// Mitsubishi GX Works2 project: GHEP-Q02U   PLC: Q02U

// global labels: Global1
VAR_GLOBAL
  Servo_Ready_T AT M1104 : BOOL;  (* Cam bien Servo Ready Truc Thu T (X0 16DT) *)
  Servo_Ready_X1 AT M1105 : BOOL;  (* Cam bien Servo Ready Truc Xa X1 (X1 16DT) *)
  Servo_Ready_X2 AT M1106 : BOOL;  (* Cam bien Servo Ready Truc Master X2 (X2 16DT) *)
  Servo_Ready_Ms AT M1107 : BOOL;  (* Cam bien Servo Ready Truc Ghep Ms (X3 16DT) *)
  Servo_Ready_S AT M1108 : BOOL;  (* Cam bien Servo Ready Truc Trang Dau S (X4 16DT) *)
  Pen1_Input_16DT AT M1109 : BOOL;  (* Tin hieu Pen 1 (X5 16DT) *)
  Pen2_Input_16DT AT M1110 : BOOL;  (* Tin hieu Pen 2 (X6 16DT) *)
  Jog_Input_16DT AT M1111 : BOOL;  (* Tin hieu Bo Cham 16DT (X7 16DT) *)
  Sensor_Rev_M AT X50 : BOOL;  (* Cam bien tiem can dem 1 vong cuon M (X50) *)
  Sensor_Rev_U AT X51 : BOOL;  (* Cam bien tiem can dem 1 vong cuon U (X51) *)
  Physical_Start_PB AT X52 : BOOL;  (* Nut nhan vat ly START QX40 (X52) *)
  Physical_Stop_PB AT X53 : BOOL;  (* Nut nhan vat ly STOP QX40 (X53) *)
  Physical_Inc_PB AT X54 : BOOL;  (* Nut nhan vat ly TANG TOC INC QX40 (X54) *)
  Physical_Dec_PB AT X55 : BOOL;  (* Nut nhan vat ly GIAM TOC DEC QX40 (X55) *)
  Pen1_Toggle_PB AT X56 : BOOL;  (* Nut nhan Toggle Pen 1 QX40 (X56) *)
  Pen2_Toggle_PB AT X57 : BOOL;  (* Nut nhan Toggle Pen 2 QX40 (X57) *)
  Switch_Hold_M AT X58 : BOOL;  (* Cong tac giu Torque Thang M khi dung (X58) *)
  Switch_Hold_U AT X59 : BOOL;  (* Cong tac giu Torque Xa U khi dung (X59) *)
  Switch_Wash_Ms AT X5A : BOOL;  (* Cong tac quay rua may bo cham Ms khi dung (X5A) *)
  Switch_Wash_S AT X5B : BOOL;  (* Cong tac quay rua may bo cham S khi dung (X5B) *)
  Physical_Jog_PB AT X5C : BOOL;  (* Nut nhan co ben ngoai BO CHAM NOI MANG QX40 (X5C) *)
  Servo_ON_T AT M1304 : BOOL;  (* Ngo ra Servo ON Truc Thu T (Y8 16DT) *)
  Servo_ON_X1 AT M1305 : BOOL;  (* Ngo ra Servo ON Truc Xa X1 (Y9 16DT) *)
  Servo_ON_X2 AT M1306 : BOOL;  (* Ngo ra Servo ON Truc Master X2 (YA 16DT) *)
  Servo_ON_Ms AT M1307 : BOOL;  (* Ngo ra Servo ON Truc Ghep Ms (YB 16DT) *)
  Servo_ON_S AT M1308 : BOOL;  (* Ngo ra Servo ON Truc Trang Dau S (YC 16DT) *)
  Pen1_Output AT M1309 : BOOL;  (* Ngo ra Ben Ep Pen 1 (YD 16DT) *)
  Pen2_Output AT M1310 : BOOL;  (* Ngo ra Ben Ep Pen 2 (YE 16DT) *)
  HMI_Auto_Mode AT M100 : BOOL;  (* Che do Auto / Manual *)
  HMI_Reset_Error AT M101 : BOOL;  (* Reset loi he thong *)
  HMI_Start AT M102 : BOOL;  (* Nut Start khoi dong HMI *)
  HMI_Stop AT M103 : BOOL;  (* Nut Stop dung may HMI *)
  HMI_Reset_Length AT M104 : BOOL;  (* Reset tong chieu dai met hang *)
  HMI_Reset_Roll_T AT M105 : BOOL;  (* Nap lai duong kinh cuon moi T *)
  HMI_Reset_Roll_M AT M106 : BOOL;  (* Nap lai duong kinh cuon moi M *)
  HMI_Reset_Roll_U AT M107 : BOOL;  (* Nap lai duong kinh cuon moi U *)
  HMI_PID_Enable AT M108 : BOOL;  (* Bat tat che do PID *)
  HMI_Inc_Hold AT M109 : BOOL;  (* Phim INC tang toc HMI *)
  HMI_Dec_Hold AT M114 : BOOL;  (* Phim DEC giam toc HMI *)
  HMI_Pen1_Cmd AT M115 : BOOL;  (* Lenh ON/OFF Pen 1 tu HMI *)
  HMI_Pen2_Cmd AT M116 : BOOL;  (* Lenh ON/OFF Pen 2 tu HMI *)
  Zero_Set_T AT M110 : BOOL;  (* Nut Set Zero Loadcell T *)
  Zero_Set_X1 AT M111 : BOOL;  (* Nut Set Zero Loadcell X1 *)
  Zero_Set_M AT M112 : BOOL;  (* Nut Set Zero Loadcell M *)
  Zero_Set_U AT M113 : BOOL;  (* Nut Set Zero Loadcell U *)
  HMI_Test_T AT M170 : BOOL;  (* Co Test chay thu rieng Truc Thu T *)
  HMI_Test_X1 AT M171 : BOOL;  (* Co Test chay thu rieng Truc Xa X1 *)
  HMI_Test_X2 AT M172 : BOOL;  (* Co Test chay thu rieng Truc Master X2 *)
  HMI_Test_Ms AT M173 : BOOL;  (* Co Test chay thu rieng Truc Ghep Ms *)
  HMI_Test_S AT M174 : BOOL;  (* Co Test chay thu rieng Truc Trang Dau S *)
  HMI_Test_M AT M175 : BOOL;  (* Co Test thu Luc Thang Tu M *)
  HMI_Test_U AT M176 : BOOL;  (* Co Test chay thu rieng Truc Xa Metalize U *)
  Calib_Set_T AT M120 : BOOL;  (* Nut Calib Span Loadcell T *)
  Calib_Set_X1 AT M121 : BOOL;  (* Nut Calib Span Loadcell X1 *)
  Calib_Set_M AT M122 : BOOL;  (* Nut Calib Span Loadcell M *)
  Calib_Set_U AT M123 : BOOL;  (* Nut Calib Span Loadcell U *)
  Servo_Not_Ready_Fault AT M134 : BOOL;  (* Co bao loi Servo Not Ready *)
  Hold_Torque_Stop_M AT M130 : BOOL;  (* Giu Torque M khi dung may *)
  Hold_Torque_Stop_U AT M131 : BOOL;  (* Giu Torque U khi dung may *)
  Anti_Dry_Rotate_S AT M132 : BOOL;  (* Bo cham S khi dung may *)
  Anti_Dry_Rotate_Ms AT M133 : BOOL;  (* Bo cham Ms khi dung may *)
  HMI_Reset_All_Rolls AT M135 : BOOL;  (* Nut thay cuon moi toan bo (Reset ca 3 cuon va xoa met) *)
  HMI_Jog_Crawl_Cmd AT M136 : BOOL;  (* Nut bo cham noi mang 2 m/p giu de chay tha de dung *)
  HMI_Cmd_Apply_Recipe AT M137 : BOOL;  (* Nut ap dung cong thuc don hang da chon *)
  HMI_Cmd_Save_Recipe AT M138 : BOOL;  (* Nut luu thong so hien tai vao cong thuc *)
  Weight_Net_T AT D510 : REAL;  (* Trong luong Luc cang thuc te T (kg/N) *)
  Weight_Net_X1 AT D512 : REAL;  (* Trong luong Luc cang thuc te X1 (kg/N) *)
  Weight_Net_M AT D514 : REAL;  (* Trong luong Luc cang thuc te M (kg/N) *)
  Weight_Net_U AT D516 : REAL;  (* Trong luong Luc cang thuc te U (kg/N) *)
  HMI_Cmd_Zero_Set AT M118 : BOOL;  (* Nut bam Set Zero chung cho truc dang chon tren HMI *)
  HMI_Cmd_Calib_Set AT M119 : BOOL;  (* Nut bam Calib Span chung cho truc dang chon tren HMI *)
  HMI_Cmd_Save_PID AT M125 : BOOL;  (* Nut bam Luu cai dat PID / Calib tren HMI *)
  HMI_Cmd_AutoTune AT M126 : BOOL;  (* Nut bam Kich hoat Auto-Tuning PID cho truc dang chon *)
  HMI_Status_AT_Busy AT M127 : BOOL;  (* Den bao dang chay Auto-Tuning *)
  HMI_Status_AT_Done AT M128 : BOOL;  (* Den bao da Auto-Tuning xong va da tu cap nhat Kp Ki Kd *)
  HMI_Status_Text_Code AT D602 : INT;  (* Ma trang thai van hanh hien thi tieng Viet tren HMI *)
  HMI_Recipe_Select AT D604 : INT;  (* Chon cong thuc don hang Recipe (1..5) *)
  HMI_Disp_Zero_Offset AT D608 : REAL;  (* O nhap Zero Offset duy nhat tren HMI *)
  HMI_Axis_Select AT D610 : INT;  (* Chon truc tren HMI (1=Thu T, 2=Xa X1, 3=Master X2, 4=Ghep Ms, 5=Dau S, 6=Thang M, 7=Xa U) *)
  HMI_Disp_Kp AT D612 : REAL;  (* O nhap Kp duy nhat tren HMI *)
  HMI_Disp_Ki AT D614 : REAL;  (* O nhap Ki duy nhat tren HMI *)
  HMI_Disp_Kd AT D616 : REAL;  (* O nhap Kd duy nhat tren HMI *)
  HMI_Disp_Calib_Gain AT D618 : REAL;  (* O nhap Calib Gain duy nhat tren HMI *)
  Gear_Ratio_T AT D620 : REAL;  (* Ty so truyen Hop so Thu T (vi du 10.1) *)
  Gear_Ratio_X1 AT D622 : REAL;  (* Ty so truyen Hop so Xa X1 (vi du 8.0) *)
  Gear_Ratio_X2 AT D624 : REAL;  (* Ty so truyen Hop so Master X2 (vi du 8.0) *)
  Gear_Ratio_Ms AT D626 : REAL;  (* Ty so truyen Hop so Ghep Ms (vi du 10.0) *)
  Gear_Ratio_S AT D628 : REAL;  (* Ty so truyen Hop so Trang Dau S (vi du 10.0) *)
  Gear_Ratio_U AT D630 : REAL;  (* Ty so truyen Hop so Xa U (vi du 1.0) *)
  Dia_X1_Roller_mm AT D638 : REAL;  (* Duong kinh lo Keo X1 (mm, vi du 300.5) *)
  Dia_Ms_Roller_mm AT D640 : REAL;  (* Duong kinh lo ghep Ms (mm, vi du 200.0) *)
  Dia_X2_Roller_mm AT D642 : REAL;  (* Duong kinh lo Master X2 (mm, vi du 300.5) *)
  Dia_S_Roller_mm AT D648 : REAL;  (* Duong kinh lo Dau S (mm, vi du 100.0) *)
  SP_Tension_T AT D660 : REAL;  (* Luc cang SP Truc T (kg) *)
  SP_Tension_X1 AT D662 : REAL;  (* Luc cang SP Truc X1 (kg) *)
  SP_Tension_M AT D664 : REAL;  (* Luc cang SP Truc M (kg) *)
  Taper_Percent_T AT D666 : REAL;  (* Ty le Con giam luc cang cuon thu T (%) *)
  SP_Tension_U AT D668 : REAL;  (* Luc cang SP Truc U (kg) *)
  Kp_T AT D670 : REAL;  (* He so Kp PID Truc T *)
  Ki_T AT D672 : REAL;  (* He so Ki PID Truc T *)
  Kd_T AT D674 : REAL;  (* He so Kd PID Truc T *)
  Kp_X1 AT D676 : REAL;  (* He so Kp PID Truc X1 *)
  Ki_X1 AT D678 : REAL;  (* He so Ki PID Truc X1 *)
  Kd_X1 AT D680 : REAL;  (* He so Kd PID Truc X1 *)
  Kp_X2 AT D682 : REAL;  (* He so Kp PID Toc do Master X2 *)
  Ki_X2 AT D684 : REAL;  (* He so Ki PID Toc do Master X2 *)
  Kd_X2 AT D686 : REAL;  (* He so Kd PID Toc do Master X2 *)
  Kp_Ms AT D688 : REAL;  (* He so Kp PID Toc do Ghep Ms *)
  Ki_Ms AT D689 : REAL;  (* He so Ki PID Toc do Ghep Ms *)
  Kd_Ms AT D692 : REAL;  (* He so Kd PID Toc do Ghep Ms *)
  Kp_S AT D694 : REAL;  (* He so Kp PID Toc do Truc S *)
  Ki_S AT D696 : REAL;  (* He so Ki PID Toc do Truc S *)
  Kd_S AT D698 : REAL;  (* He so Kd PID Toc do Truc S *)
  Set_Target_Length AT D700 : REAL;  (* Chieu dai met hang cai dat tu dung (m) *)
  Decel_Distance_Meters AT D702 : REAL;  (* Khoang cach bao giam toc truoc khi dung (m) *)
  Ramp_Accel_Rate AT D704 : REAL;  (* Thanh ghi gia toc ACC (m/p/s) *)
  Ramp_Decel_Rate AT D706 : REAL;  (* Thanh ghi giam toc DEC (m/p/s) *)
  Total_Length_Meters AT D708 : REAL;  (* Tong so met hang da ghep (m) *)
  Release_Pen_Speed_MPM AT D710 : REAL;  (* Toc do nhan bi 2 Pen ep mang (m/p) *)
  Real_Dia_U_mm AT D720 : REAL;  (* Duong kinh thuc cuon U (mm) *)
  Real_Dia_M_mm AT D722 : REAL;  (* Duong kinh thuc cuon M (mm) *)
  Real_Dia_T_mm AT D724 : REAL;  (* Duong kinh thuc cuon T (mm) *)
  Current_Line_MPM AT D730 : REAL;  (* Toc do hien tai (m/p) *)
  Target_Line_MPM AT D732 : REAL;  (* Toc do muc tieu (m/p) *)
  Max_Speed_MPM AT D734 : REAL;  (* Toc do Max (100.0 m/p) *)
  Min_Speed_MPM AT D736 : REAL;  (* Toc do Min (2.0 m/p) *)
  Anti_Dry_Crawl_Speed AT D738 : REAL;  (* Toc do bo cham rua may (1.0 m/p) *)
  Core_Dia_T_mm AT D740 : REAL;  (* Duong kinh loi cuon T (mm) *)
  Core_Dia_M_mm AT D742 : REAL;  (* Duong kinh loi cuon M (mm) *)
  Core_Dia_U_mm AT D744 : REAL;  (* Duong kinh loi cuon U (mm) *)
  Max_Dia_T_mm AT D750 : REAL;  (* Duong kinh Max cuon T (mm) *)
  Max_Dia_M_mm AT D752 : REAL;  (* Duong kinh Max cuon M (mm) *)
  Max_Dia_U_mm AT D754 : REAL;  (* Duong kinh Max cuon U (mm) *)
  Speed_Ratio_T AT D756 : REAL;  (* Ty le toc do Truc T giu Torque (vi du 1.05) *)
  Speed_Ratio_X1 AT D758 : REAL;  (* Ty le toc do Truc Xa X1 (vi du 1.00) *)
  Speed_Offset_X1 AT D760 : REAL;  (* Bu toc do Truc Xa X1 *)
  Speed_Ratio_Ms AT D762 : REAL;  (* Ty le dong bo toc do Truc Ms (vi du 1.00) *)
  Speed_Offset_Ms AT D764 : REAL;  (* Bu toc do Truc Ghep Ms *)
  Speed_Ratio_S AT D766 : REAL;  (* Ty le toc do Truc S (vi du 1.00) *)
  Speed_Offset_S AT D768 : REAL;  (* Bu toc do Truc Trang Dau S *)
  Min_Torque_M AT D770 : REAL;  (* Torque Min Thang M (%) *)
  Max_Torque_M AT D772 : REAL;  (* Torque Max Thang M (%) *)
  Init_Holding_Torque_M AT D774 : REAL;  (* Torque ban dau Thang M (%) *)
  Init_Holding_Torque_U AT D776 : REAL;  (* Torque ban dau giu cuon U (%) *)
  Min_Torque_U AT D778 : REAL;  (* Torque Min Xa U (%) *)
  Max_Torque_U AT D780 : REAL;  (* Torque Max Xa U (%) *)
  SP_Speed_S AT D782 : REAL;  (* Toc do Setpoint Truc S *)
  Feedback_Speed_S AT D784 : REAL;  (* Toc do Feedback Truc S *)
  Feedback_Speed_X2 AT D786 : REAL;  (* Toc do Feedback Master X2 *)
  Feedback_Speed_Ms AT D788 : REAL;  (* Toc do Feedback Ghep Ms *)
  Test_Speed_T AT D800 : REAL;  (* Toc do cai dat Test Truc T (0..16000) *)
  Test_Torque_T AT D802 : REAL;  (* Torque cai dat Test Truc T (0..16000) *)
  Test_Speed_X1 AT D804 : REAL;  (* Toc do cai dat Test Truc X1 (0..16000) *)
  Test_Speed_X2 AT D806 : REAL;  (* Toc do cai dat Test Truc X2 (0..16000) *)
  Test_Speed_Ms AT D808 : REAL;  (* Toc do cai dat Test Truc Ms (0..16000) *)
  Test_Speed_S AT D810 : REAL;  (* Toc do cai dat Test Truc S (0..16000) *)
  Test_Torque_M AT D812 : REAL;  (* Torque cai dat Test Thang M (0..16000) *)
  Test_Speed_U AT D814 : REAL;  (* Toc do cai dat Test Truc U (0..16000) *)
  Max_RPM_X2 AT D820 : REAL;  (* Toc do Max RPM Master X2 (1000.0) *)
  Max_RPM_X1 AT D822 : REAL;  (* Toc do Max RPM Xa X1 (1000.0) *)
  Max_RPM_Ms AT D824 : REAL;  (* Toc do Max RPM Ghep Ms (3000.0) *)
  Max_RPM_S AT D826 : REAL;  (* Toc do Max RPM Trang Dau S (3000.0) *)
  Max_RPM_T AT D828 : REAL;  (* Toc do Max RPM Thu T (1500.0) *)
  Calib_Gain_T AT D830 : REAL;  (* He so Calib Gain Loadcell T *)
  Calib_Gain_X1 AT D832 : REAL;  (* He so Calib Gain Loadcell X1 *)
  Calib_Gain_M AT D834 : REAL;  (* He so Calib Gain Loadcell M *)
  Calib_Gain_U AT D836 : REAL;  (* He so Calib Gain Loadcell U *)
  Kp_M AT D840 : REAL;  (* He so Kp PID Truc M *)
  Ki_M AT D842 : REAL;  (* He so Ki PID Truc M *)
  Kd_M AT D844 : REAL;  (* He so Kd PID Truc M *)
  Kp_U AT D846 : REAL;  (* He so Kp PID Truc U *)
  Ki_U AT D848 : REAL;  (* He so Ki PID Truc U *)
  Kd_U AT D850 : REAL;  (* He so Kd PID Truc U *)
  Zero_Offset_T AT D852 : REAL;  (* Diem 0 Zero Offset Loadcell Thu T *)
  Zero_Offset_X1 AT D854 : REAL;  (* Diem 0 Zero Offset Loadcell Xa X1 *)
  Zero_Offset_M AT D856 : REAL;  (* Diem 0 Zero Offset Thang Tu Metalize M *)
  Zero_Offset_U AT D858 : REAL;  (* Diem 0 Zero Offset Cuon Xa Sau Cung U *)
  CCLink_AD_Avg_Mode AT D860 : WORD;  (* Che do lay trung binh BFM 0 64AD (H3333=Moving Avg) *)
  CCLink_AD_Avg_CH1 AT D861 : INT;  (* So mau trung binh CH1 BFM 1 (Loadcell Thu T) *)
  CCLink_AD_Avg_CH2 AT D862 : INT;  (* So mau trung binh CH2 BFM 2 (Loadcell Xa X1) *)
  CCLink_AD_Avg_CH3 AT D863 : INT;  (* So mau trung binh CH3 BFM 3 (Loadcell Thang M) *)
  CCLink_AD_Avg_CH4 AT D864 : INT;  (* So mau trung binh CH4 BFM 4 (Loadcell Xa U) *)
  CCLink_AD_Conv_En AT D865 : INT;  (* Cho phep chuyen doi AD 4 kenh BFM 10 (0=Enable) *)
END_VAR

// task Task_01 (event TRUE, interval 0, priority 31): POU_01
// task POU_INIT (event TRUE, interval 0, priority 31): POU_INIT

PROGRAM POU_01
VAR
  pid_T : FB_TENSION_PID;  (* Instance PID Luc cang Thu T *)
  pid_X1 : FB_TENSION_PID;  (* Instance PID Luc cang Xa X1 *)
  pid_M : FB_TENSION_PID;  (* Instance PID Thang Tu M *)
  pid_U : FB_TENSION_PID;  (* Instance PID Luc cang Xa U *)
  pid_X2 : FB_TENSION_PID;  (* Instance PID Toc do Master X2 *)
  pid_Ms : FB_TENSION_PID;  (* Instance PID Toc do Ghep Ms *)
  pid_S : FB_TENSION_PID;  (* Instance PID Toc do Trang Dau S *)
  fbCCLink : FFB_CCLINK_CONTROL;  (* Instance Control CC-Link Master *)
  Base_Speed_X2 : REAL;  (* Toc do nen Master X2 *)
  SP_Speed_X2 : REAL;  (* Toc do Setpoint Master X2 *)
  SP_Speed_X1 : REAL;  (* Toc do Setpoint Xa X1 *)
  SP_Speed_Ms : REAL;  (* Toc do Setpoint Ghep Ms *)
  SP_Speed_T : REAL;  (* Toc do Setpoint Thu T *)
  Calc_Speed_X2 : REAL;  (* Toc do tinh toan Master X2 *)
  Calc_Speed_T : REAL;  (* Toc do tinh toan Thu T *)
  Calc_Torque_T : REAL;  (* Torque tinh toan Thu T *)
  Calc_Speed_X1 : REAL;  (* Toc do tinh toan Xa X1 *)
  Calc_Speed_Ms : REAL;  (* Toc do tinh toan Ghep Ms *)
  Calc_Speed_S : REAL;  (* Toc do tinh toan Trang Dau S *)
  Calc_Speed_U : REAL;  (* Toc do tinh toan Xa U *)
  Calc_Torque_M : REAL;  (* Torque tinh toan Thang M *)
  Base_Torque_M : REAL;  (* Torque nen co ban Thang M *)
  State_Machine : DINT;  (* Trang thai van hanh State Machine *)
  ADC_CH1_Val : WORD;  (* Bien tam doc ADC CH1 *)
  ADC_CH2_Val : WORD;  (* Bien tam doc ADC CH2 *)
  ADC_CH3_Val : WORD;  (* Bien tam doc ADC CH3 *)
  ADC_CH4_Val : WORD;  (* Bien tam doc ADC CH4 *)
  Effective_SP_T : REAL;  (* Luc cang SP cuon T sau khi tinh Con luc Taper *)
  Auto_Decel_Flag : BOOL;  (* Co tu dong giam toc khi sap dat tong chieu dai *)
  ADC_Filter_T : REAL;  (* Bo loc nhieu trung binh dong Loadcell T *)
  ADC_Filter_X1 : REAL;  (* Bo loc nhieu trung binh dong Loadcell X1 *)
  ADC_Filter_M : REAL;  (* Bo loc nhieu trung binh dong Loadcell M *)
  ADC_Filter_U : REAL;  (* Bo loc nhieu trung binh dong Loadcell U *)
  Cmd_Start : BOOL;  (* Lenh Tong Start (HMI + Nut vat ly X52) *)
  Cmd_Stop : BOOL;  (* Lenh Tong Stop (HMI + Nut vat ly X53) *)
  Cmd_Inc : BOOL;  (* Lenh Tong INC Tang toc (HMI + Nut vat ly X54) *)
  Cmd_Dec : BOOL;  (* Lenh Tong DEC Giam toc (HMI + Nut vat ly X55) *)
  Cmd_Jog_Crawl : BOOL;  (* Lenh Tong Bo cham noi mang 2 m/p (HMI + Nut co X5C) *)
  Inc_Hold_Timer : DINT;  (* Timer bam giu phim Tang toc INC *)
  Dec_Hold_Timer : DINT;  (* Timer bam giu phim Giam toc DEC *)
  Curr_Pulse_T : DINT;  (* Xung Encoder Thu T *)
  Last_Pulse_T : DINT;  (* Xung Encoder Thu T vong truoc *)
  Curr_Pulse_X2 : DINT;  (* Xung Encoder Master X2 *)
  Last_Pulse_X2_T : DINT;  (* Xung Master X2 khi Thu T quay 1 vong *)
  Last_Pulse_X2_M : DINT;  (* Xung Master X2 khi Cuon M quay 1 vong *)
  Last_Pulse_X2_U : DINT;  (* Xung Master X2 khi Cuon U quay 1 vong *)
  Last_Pulse_X2_Len : DINT;  (* Xung Master X2 vong truoc de do met *)
  Delta_Pulse_X2 : DINT;  (* So xung Master X2 tang them moi chu ky *)
  Delta_Length_mm : REAL;  (* So mm mang tang them moi chu ky *)
  Accum_Length_mm : REAL;  (* Tich luy mm mang de doi ra met *)
  Trig_X50 : BOOL;  (* Xung phat hien cam bien X50 cuon M *)
  Trig_X51 : BOOL;  (* Xung phat hien cam bien X51 cuon U *)
  Prev_X50 : BOOL;  (* Trang thai X50 vong scan truoc *)
  Prev_X51 : BOOL;  (* Trang thai X51 vong scan truoc *)
  Raw_Dia_T_mm : REAL;  (* Duong kinh tho tinh duoc cuon T *)
  Raw_Dia_M_mm : REAL;  (* Duong kinh tho tinh duoc cuon M *)
  Raw_Dia_U_mm : REAL;  (* Duong kinh tho tinh duoc cuon U *)
  Rev_Count_T : DINT;  (* So vong quay cuon T *)
  Rev_Count_M : DINT;  (* So vong quay cuon M *)
  Rev_Count_U : DINT;  (* So vong quay cuon U *)
  Dynamic_Accel_Step : REAL;  (* Buoc gia toc dong tang giam luy tien *)
  Trig_Pen1 : BOOL;  (* Xung nhan phim Toggle Pen 1 X56 *)
  Trig_Pen2 : BOOL;  (* Xung nhan phim Toggle Pen 2 X57 *)
  Prev_Pen1_PB : BOOL;  (* Trang thai X56 vong scan truoc *)
  Prev_Pen2_PB : BOOL;  (* Trang thai X57 vong scan truoc *)
  Prev_Pen1_16DT : BOOL;  (* Trang thai Pen 1 tren 16DT vong truoc *)
  Prev_Pen2_16DT : BOOL;  (* Trang thai Pen 2 tren 16DT vong truoc *)
  Pen1_State : BOOL;  (* Trang thai ON/OFF hien tai Pen 1 *)
  Pen2_State : BOOL;  (* Trang thai ON/OFF hien tai Pen 2 *)
  PID_Out_T : REAL;  (* Output PID sau khi lay tu pid_T *)
  PID_Out_X1 : REAL;  (* Output PID sau khi lay tu pid_X1 *)
  PID_Out_M : REAL;  (* Output PID sau khi lay tu pid_M *)
  PID_Out_U : REAL;  (* Output PID sau khi lay tu pid_U *)
  PID_Out_X2 : REAL;  (* Output PID Toc do X2 *)
  PID_Out_Ms : REAL;  (* Output PID Toc do Ms *)
  PID_Out_S : REAL;  (* Output PID Toc do S *)
  Trig_PID_10ms : BOOL;  (* Xung kich hoat PID moi 10ms (SM409) *)
  Prev_SM409 : BOOL;  (* Trang thai SM409 vong scan truoc *)
  Pen_Auto_Engaged : BOOL;  (* Co tu dong kep 2 Pen khi toc do vuot 5 m/p *)
  Prev_Recipe_Select : INT;  (* Luu gia tri Recipe da chon vong scan truoc *)
END_VAR
(* ============================================================================ *)
(* MÃ NGUỒN POU_01: HỆ THỐNG MÁY GHÉP MÀNG METALIZE TỰ ĐỘNG - MITSUBISHI Q02U  *)
(* ĐỒNG BỘ VẬN TỐC DÀI THEO TRỤC CHÍNH X2 + SPEED_RATIO CHO TỪNG TRỤC           *)
(* TOÀN BỘ TÍNH TOÁN DÙNG CHUẨN SỐ THỰC FLOAT / REAL (FLOAT [Single Precision]) *)
(* ============================================================================ *)

(* 1. BẢO VỆ 5 TRỤC SERVO READY TRÊN MODULE 16DT (X0..X4 = M1136..M1140 - TRẠM 5) *)
Servo_Not_Ready_Fault := NOT(Servo_Ready_T) OR NOT(Servo_Ready_X1) OR NOT(Servo_Ready_X2) OR NOT(Servo_Ready_Ms) OR NOT(Servo_Ready_S);

IF Servo_Not_Ready_Fault AND State_Machine = 1 THEN
    State_Machine := 0; (* Dừng khẩn cấp nếu đang chạy tự động *)
END_IF;

(* 2. ĐIỀU KHIỂN CÔNG TẮC GIỮ TORQUE & BÒ CHẬM RỬA MÁY TRÊN QX40 (X58..X5B) *)
Hold_Torque_Stop_M := Switch_Hold_M;   (* X58 *)
Hold_Torque_Stop_U := Switch_Hold_U;   (* X59 *)
Anti_Dry_Rotate_Ms := Switch_Wash_Ms;  (* X5A *)
Anti_Dry_Rotate_S  := Switch_Wash_S;   (* X5B *)

(* 2.1 QUẢN LÝ CÔNG THỨC ĐƠN HÀNG (RECIPE MANAGEMENT CHO CÔNG NHÂN) *)
(* 1: Màng Mỏng 12~15mic | 2: Màng Tiêu Chuẩn 18~20mic | 3: Giấy Dày Duplex 250~350g | 4: Màng Nhôm Foil | 5: Tùy Chỉnh *)
IF HMI_Recipe_Select <= 0 OR HMI_Recipe_Select > 5 THEN
    HMI_Recipe_Select := 2; (* Mặc định chọn Recipe 2: Hàng Tiêu Chuẩn *)
END_IF;

(* TỰ ĐỘNG NẠP THÔNG SỐ KHI CÔNG NHÂN CHỌN LOẠI HÀNG HOẶC NHẤN ÁP DỤNG *)
IF (HMI_Recipe_Select <> Prev_Recipe_Select) OR HMI_Cmd_Apply_Recipe THEN
    CASE HMI_Recipe_Select OF
        1: (* 1. HÀNG MÀNG MỎNG (BOPP 12~15 mic - Bao bì bánh kẹo) *)
            Target_Line_MPM  := 45.0;  (* Tốc độ chuẩn 45 m/p *)
            SP_Tension_T     := 12.0;  (* Lực căng Thu T: 12 kg *)
            SP_Tension_X1    := 10.0;  (* Lực căng Kéo X1: 10 kg *)
            SP_Tension_M     := 4.0;   (* Lực căng Thắng Metalize M: 4 kg *)
            SP_Tension_U     := 8.0;   (* Lực căng Xả U: 8 kg *)
            Taper_Percent_T  := 15.0;  (* Giảm côn lực 15% *)
            Ramp_Accel_Rate  := 0.05;  (* Gia tốc êm ái *)
            Ramp_Decel_Rate  := 0.08;

        2: (* 2. HÀNG TIÊU CHUẨN (BOPP 18~20 mic + Giấy 100~150g - Hộp thông dụng) *)
            Target_Line_MPM  := 60.0;  (* Tốc độ chuẩn 60 m/p *)
            SP_Tension_T     := 16.0;  (* Lực căng Thu T: 16 kg *)
            SP_Tension_X1    := 14.0;  (* Lực căng Kéo X1: 14 kg *)
            SP_Tension_M     := 6.0;   (* Lực căng Thắng Metalize M: 6 kg *)
            SP_Tension_U     := 12.0;  (* Lực căng Xả U: 12 kg *)
            Taper_Percent_T  := 20.0;  (* Giảm côn lực 20% *)
            Ramp_Accel_Rate  := 0.08;  (* Gia tốc tiêu chuẩn *)
            Ramp_Decel_Rate  := 0.10;

        3: (* 3. HÀNG GIẤY DÀY / BÌA CỨNG (Duplex / Ivory 250~350g + Metalize) *)
            Target_Line_MPM  := 50.0;  (* Tốc độ chuẩn 50 m/p *)
            SP_Tension_T     := 25.0;  (* Lực căng Thu T: 25 kg *)
            SP_Tension_X1    := 22.0;  (* Lực căng Kéo X1: 22 kg *)
            SP_Tension_M     := 8.0;   (* Lực căng Thắng Metalize M: 8 kg *)
            SP_Tension_U     := 18.0;  (* Lực căng Xả U: 18 kg *)
            Taper_Percent_T  := 25.0;  (* Giảm côn lực 25% *)
            Ramp_Accel_Rate  := 0.06;
            Ramp_Decel_Rate  := 0.10;

        4: (* 4. HÀNG MÀNG NHÔM / FOIL DẺO CAO CẤP (Alu Foil 9~12 mic / PET) *)
            Target_Line_MPM  := 40.0;  (* Tốc độ chuẩn 40 m/p *)
            SP_Tension_T     := 10.0;  (* Lực căng Thu T: 10 kg *)
            SP_Tension_X1    := 8.0;   (* Lực căng Kéo X1: 8 kg *)
            SP_Tension_M     := 3.5;   (* Lực căng Thắng Metalize M: 3.5 kg *)
            SP_Tension_U     := 7.0;   (* Lực căng Xả U: 7 kg *)
            Taper_Percent_T  := 15.0;
            Ramp_Accel_Rate  := 0.04;  (* Gia tốc siêu êm chống đứt foil *)
            Ramp_Decel_Rate  := 0.06;

        5: (* 5. CHẾ ĐỘ TÙY CHỈNH (CUSTOM) *)
            Target_Line_MPM := Target_Line_MPM; (* Giữ nguyên thông số người dùng tùy chỉnh *)
    END_CASE;
    Prev_Recipe_Select   := HMI_Recipe_Select;
    HMI_Cmd_Apply_Recipe := FALSE;
END_IF;

IF HMI_Cmd_Save_Recipe THEN
    HMI_Recipe_Select    := 5;
    Prev_Recipe_Select   := 5;
    HMI_Cmd_Save_Recipe  := FALSE;
END_IF;

(* 3. NẠP LẠI ĐƯỜNG KÍNH CUỘN TỪ HMI & NÚT THAY CUỘN MỚI TOÀN BỘ 1-CLICK *)
IF HMI_Reset_All_Rolls THEN
    Real_Dia_T_mm       := Core_Dia_T_mm; (* Thu T về lõi *)
    Real_Dia_M_mm       := Max_Dia_M_mm;  (* Thắng M về cuộn đầy *)
    Real_Dia_U_mm       := Max_Dia_U_mm;  (* Xả U về cuộn đầy *)
    Total_Length_Meters := 0.0;           (* Xóa mét về 0 *)
    Accum_Length_mm     := 0.0;
    HMI_Reset_All_Rolls := FALSE;
END_IF;
IF HMI_Reset_Roll_T THEN Real_Dia_T_mm := Core_Dia_T_mm; HMI_Reset_Roll_T := FALSE; END_IF;
IF HMI_Reset_Roll_M THEN Real_Dia_M_mm := Max_Dia_M_mm;  HMI_Reset_Roll_M := FALSE; END_IF;
IF HMI_Reset_Roll_U THEN Real_Dia_U_mm := Max_Dia_U_mm;  HMI_Reset_Roll_U := FALSE; END_IF;

(* 4. TỔNG HỢP NÚT NHẤN HMI & NÚT NHẤN VẬT LÝ TRÊN QX40 (X52..X55, X5C) *)
Cmd_Start     := HMI_Start OR Physical_Start_PB;
Cmd_Stop      := HMI_Stop OR Physical_Stop_PB OR Servo_Not_Ready_Fault;
Cmd_Inc       := HMI_Inc_Hold OR Physical_Inc_PB;
Cmd_Dec       := HMI_Dec_Hold OR Physical_Dec_PB;
Cmd_Jog_Crawl := HMI_Jog_Crawl_Cmd OR Physical_Jog_PB OR Jog_Input_16DT;

(* 5. ĐIỀU KHIỂN TOGGLE 2 PEN ÉP MÀNG (QX40 X56/X57 HOẶC 16DT X5/X6) *)
Trig_Pen1 := (Pen1_Toggle_PB AND NOT(Prev_Pen1_PB)) OR (Pen1_Input_16DT AND NOT(Prev_Pen1_16DT)) OR HMI_Pen1_Cmd;
Prev_Pen1_PB := Pen1_Toggle_PB;
Prev_Pen1_16DT := Pen1_Input_16DT;
IF HMI_Pen1_Cmd THEN HMI_Pen1_Cmd := FALSE; END_IF;
IF Trig_Pen1 THEN Pen1_State := NOT(Pen1_State); END_IF;

Trig_Pen2 := (Pen2_Toggle_PB AND NOT(Prev_Pen2_PB)) OR (Pen2_Input_16DT AND NOT(Prev_Pen2_16DT)) OR HMI_Pen2_Cmd;
Prev_Pen2_PB := Pen2_Toggle_PB;
Prev_Pen2_16DT := Pen2_Input_16DT;
IF HMI_Pen2_Cmd THEN HMI_Pen2_Cmd := FALSE; END_IF;
IF Trig_Pen2 THEN Pen2_State := NOT(Pen2_State); END_IF;

(* TỰ ĐỘNG ĐÓNG 2 PEN KHI TỐC ĐỘ VƯỢT 5.0 m/p VÀ TỰ ĐỘNG NHẢ KHI DỪNG / DƯỚI RELEASE SPEED *)
IF State_Machine = 1 AND Current_Line_MPM >= 5.0 AND NOT(Pen_Auto_Engaged) THEN
    Pen1_State := TRUE;
    Pen2_State := TRUE;
    Pen_Auto_Engaged := TRUE;
ELSIF State_Machine = 0 OR Current_Line_MPM <= Release_Pen_Speed_MPM THEN
    Pen1_State := FALSE;
    Pen2_State := FALSE;
    Pen_Auto_Engaged := FALSE;
END_IF;

M1309 := Pen1_State; (* YD trên 16DT: Van Solenoid Pen 1 *)
M1310 := Pen2_State; (* YE trên 16DT: Van Solenoid Pen 2 *)

(* 6. TĂNG GIẢM TỐC LŨY TIẾN THEO THỜI GIAN GIỮ PHÍM INC / DEC *)
IF Cmd_Inc THEN
    Inc_Hold_Timer := Inc_Hold_Timer + 1;
    IF Inc_Hold_Timer < 50 THEN
        Dynamic_Accel_Step := Ramp_Accel_Rate;
    ELSIF Inc_Hold_Timer < 150 THEN
        Dynamic_Accel_Step := Ramp_Accel_Rate * 2.0;
    ELSE
        Dynamic_Accel_Step := Ramp_Accel_Rate * 5.0;
    END_IF;
    Target_Line_MPM := Target_Line_MPM + Dynamic_Accel_Step;
    IF Target_Line_MPM > Max_Speed_MPM THEN Target_Line_MPM := Max_Speed_MPM; END_IF;
ELSE
    Inc_Hold_Timer := 0;
END_IF;

IF Cmd_Dec THEN
    Dec_Hold_Timer := Dec_Hold_Timer + 1;
    IF Dec_Hold_Timer < 50 THEN
        Dynamic_Accel_Step := Ramp_Decel_Rate;
    ELSIF Dec_Hold_Timer < 150 THEN
        Dynamic_Accel_Step := Ramp_Decel_Rate * 2.0;
    ELSE
        Dynamic_Accel_Step := Ramp_Decel_Rate * 5.0;
    END_IF;
    Target_Line_MPM := Target_Line_MPM - Dynamic_Accel_Step;
    IF Target_Line_MPM < Min_Speed_MPM THEN Target_Line_MPM := Min_Speed_MPM; END_IF;
ELSE
    Dec_Hold_Timer := 0;
END_IF;

(* RAMPING TỐC ĐỘ HIỆN TẠI (FLOAT) *)
IF Current_Line_MPM < Target_Line_MPM THEN
    Current_Line_MPM := Current_Line_MPM + Ramp_Accel_Rate;
    IF Current_Line_MPM > Target_Line_MPM THEN Current_Line_MPM := Target_Line_MPM; END_IF;
ELSIF Current_Line_MPM > Target_Line_MPM THEN
    Current_Line_MPM := Current_Line_MPM - Ramp_Decel_Rate;
    IF Current_Line_MPM < Target_Line_MPM THEN Current_Line_MPM := Target_Line_MPM; END_IF;
END_IF;

(* 7. TÍNH ĐƯỜNG KÍNH 3 CUỘN T, M, U VÀ ĐO CHIỀU DÀI MÀNG CHẠY *)
Curr_Pulse_T  := INT_TO_DINT(WORD_TO_INT(D5000));
Curr_Pulse_X2 := INT_TO_DINT(WORD_TO_INT(D5002));

(* TÍNH TOÁN CHIỀU DÀI MÀNG CHẠY TÍCH LŨY TỪ XUNG ENCODER MASTER X2 *)
IF Curr_Pulse_X2 >= Last_Pulse_X2_Len THEN
    Delta_Pulse_X2 := Curr_Pulse_X2 - Last_Pulse_X2_Len;
ELSE
    Delta_Pulse_X2 := (Curr_Pulse_X2 + 65536) - Last_Pulse_X2_Len;
END_IF;

IF Delta_Pulse_X2 > 0 AND State_Machine = 1 AND Gear_Ratio_X2 > 0.0 THEN
    (* Chu vi Lô X2 = PI * Dia_X2_Roller_mm *)
    (* Delta_Length = Delta_Pulse_X2 * (PI * Dia_X2_Roller_mm) / (8000.0 * Gear_Ratio_X2) *)
    Delta_Length_mm := (DINT_TO_REAL(Delta_Pulse_X2) * 3.1415 * Dia_X2_Roller_mm) / (8000.0 * Gear_Ratio_X2);
    Accum_Length_mm := Accum_Length_mm + Delta_Length_mm;
    
    (* Chuyển đổi mm sang mét *)
    IF Accum_Length_mm >= 1000.0 THEN
        Total_Length_Meters := Total_Length_Meters + (Accum_Length_mm / 1000.0);
        Accum_Length_mm     := 0.0;
    END_IF;
END_IF;
Last_Pulse_X2_Len := Curr_Pulse_X2;

(* NÚT RESET TỔNG CHIỀU DÀI MÉT TỪ HMI (M104) *)
IF HMI_Reset_Length THEN
    Total_Length_Meters := 0.0;
    Accum_Length_mm     := 0.0;
    HMI_Reset_Length    := FALSE;
END_IF;

(* TÍNH ĐƯỜNG KÍNH CUỘN THU T THEO XUNG MASTER X2 (1 VÒNG THU T = 8000 * Gear_Ratio_T) *)
IF Gear_Ratio_T > 0.0 AND (Curr_Pulse_T - Last_Pulse_T) >= REAL_TO_DINT(8000.0 * Gear_Ratio_T) THEN
    Rev_Count_T := Rev_Count_T + 1;
    IF (Curr_Pulse_X2 - Last_Pulse_X2_T) > 0 AND Gear_Ratio_X2 > 0.0 THEN
        Raw_Dia_T_mm := (DINT_TO_REAL(Curr_Pulse_X2 - Last_Pulse_X2_T) * Dia_X2_Roller_mm) / (8000.0 * Gear_Ratio_X2);
        IF Raw_Dia_T_mm < Core_Dia_T_mm THEN Raw_Dia_T_mm := Core_Dia_T_mm; END_IF;
        IF Raw_Dia_T_mm > Max_Dia_T_mm THEN Raw_Dia_T_mm := Max_Dia_T_mm; END_IF;
        Real_Dia_T_mm := Real_Dia_T_mm + ((Raw_Dia_T_mm - Real_Dia_T_mm) * 0.2);
    END_IF;
    Last_Pulse_X2_T := Curr_Pulse_X2;
    Last_Pulse_T    := Curr_Pulse_T;
END_IF;

(* TÍNH ĐƯỜNG KÍNH CUỘN XẢ M THEO CẢM BIẾN TIỆM CẬN X50 *)
Trig_X50 := Sensor_Rev_M AND NOT(Prev_X50);
Prev_X50 := Sensor_Rev_M;
IF Trig_X50 THEN
    Rev_Count_M := Rev_Count_M + 1;
    IF (Curr_Pulse_X2 - Last_Pulse_X2_M) > 0 AND Gear_Ratio_X2 > 0.0 THEN
        Raw_Dia_M_mm := (DINT_TO_REAL(Curr_Pulse_X2 - Last_Pulse_X2_M) * Dia_X2_Roller_mm) / (8000.0 * Gear_Ratio_X2);
        IF Raw_Dia_M_mm < Core_Dia_M_mm THEN Raw_Dia_M_mm := Core_Dia_M_mm; END_IF;
        IF Raw_Dia_M_mm > Max_Dia_M_mm THEN Raw_Dia_M_mm := Max_Dia_M_mm; END_IF;
        Real_Dia_M_mm := Real_Dia_M_mm + ((Raw_Dia_M_mm - Real_Dia_M_mm) * 0.2);
    END_IF;
    Last_Pulse_X2_M := Curr_Pulse_X2;
END_IF;

(* TÍNH ĐƯỜNG KÍNH CUỘN XẢ U THEO CẢM BIẾN TIỆM CẬN X51 *)
Trig_X51 := Sensor_Rev_U AND NOT(Prev_X51);
Prev_X51 := Sensor_Rev_U;
IF Trig_X51 THEN
    Rev_Count_U := Rev_Count_U + 1;
    IF (Curr_Pulse_X2 - Last_Pulse_X2_U) > 0 AND Gear_Ratio_X2 > 0.0 THEN
        Raw_Dia_U_mm := (DINT_TO_REAL(Curr_Pulse_X2 - Last_Pulse_X2_U) * Dia_X2_Roller_mm) / (8000.0 * Gear_Ratio_X2);
        IF Raw_Dia_U_mm < Core_Dia_U_mm THEN Raw_Dia_U_mm := Core_Dia_U_mm; END_IF;
        IF Raw_Dia_U_mm > Max_Dia_U_mm THEN Raw_Dia_U_mm := Max_Dia_U_mm; END_IF;
        Real_Dia_U_mm := Real_Dia_U_mm + ((Raw_Dia_U_mm - Real_Dia_U_mm) * 0.2);
    END_IF;
    Last_Pulse_X2_U := Curr_Pulse_X2;
END_IF;

(* 8. STATE MACHINE VẬN HÀNH DÂY CHUYỀN & CHẾ ĐỘ BÒ CHẬM NỐI MÀNG *)
CASE State_Machine OF
    0: (* STATE_STOPPED *)
        IF Cmd_Jog_Crawl AND NOT(Servo_Not_Ready_Fault) THEN
            (* Chế độ bò chậm 2.0 m/phút để luồn nối màng từ nút cơ ngoài X5C hoặc HMI *)
            Target_Line_MPM := Min_Speed_MPM;
            IF Target_Line_MPM <= 0.0 THEN Target_Line_MPM := 2.0; END_IF;
        ELSE
            Current_Line_MPM := 0.0;
            Target_Line_MPM  := 0.0;
        END_IF;

        IF Cmd_Start AND NOT(Servo_Not_Ready_Fault) THEN
            State_Machine   := 1;
            HMI_PID_Enable  := TRUE; (* Tự động kích hoạt PID cho công nhân *)
            HMI_Start       := FALSE;
            IF Target_Line_MPM < Min_Speed_MPM THEN Target_Line_MPM := 20.0; END_IF;
        END_IF;

    1: (* STATE_RUNNING *)
        IF Cmd_Stop THEN
            State_Machine := 0;
            HMI_Stop := FALSE;
        END_IF;
END_CASE;

(* ĐIỀU KHIỂN 5 TRỤC SERVO ON XUẤT RA MODULE 16DT (Y8..YC = M1304..M1308) *)
M1304 := (State_Machine = 1) OR HMI_Test_T;
M1305 := (State_Machine = 1) OR HMI_Test_X1;
M1306 := (State_Machine = 1) OR HMI_Test_X2;
M1307 := (State_Machine = 1) OR HMI_Test_Ms OR (State_Machine = 0 AND Anti_Dry_Rotate_Ms);
M1308 := (State_Machine = 1) OR HMI_Test_S  OR (State_Machine = 0 AND Anti_Dry_Rotate_S);

Servo_ON_T  := M1304;
Servo_ON_X1 := M1305;
Servo_ON_X2 := M1306;
Servo_ON_Ms := M1307;
Servo_ON_S  := M1308;

(* 9. TÍNH CÔN LỰC TAPER TENSION CUỘN THU T (FLOAT) *)
IF (Max_Dia_T_mm - Core_Dia_T_mm) > 0.0 AND Taper_Percent_T > 0.0 THEN
    Effective_SP_T := SP_Tension_T - (((Real_Dia_T_mm - Core_Dia_T_mm) * SP_Tension_T * (Taper_Percent_T / 100.0)) / (Max_Dia_T_mm - Core_Dia_T_mm));
ELSE
    Effective_SP_T := SP_Tension_T;
END_IF;
IF Effective_SP_T < 0.0 THEN Effective_SP_T := 0.0; END_IF;

(* TÍNH TOÁN TỐC ĐỘ ĐẶT SETPOINT CHO CÁC TRỤC ĐỒNG BỘ THEO MASTER X2 (HIGH RESOLUTION 0..16000) *)
IF Max_Speed_MPM > 0.0 THEN
    Base_Speed_X2 := (Current_Line_MPM * 16000.0) / Max_Speed_MPM;
ELSE
    Base_Speed_X2 := 0.0;
END_IF;

SP_Speed_X2 := Base_Speed_X2;
SP_Speed_X1 := (Base_Speed_X2 * Speed_Ratio_X1) + Speed_Offset_X1;

IF Dia_X2_Roller_mm > 0.0 THEN
    SP_Speed_Ms := (((Base_Speed_X2 * Dia_Ms_Roller_mm) / Dia_X2_Roller_mm) * Speed_Ratio_Ms) + Speed_Offset_Ms;
ELSE
    SP_Speed_Ms := Base_Speed_X2 + Speed_Offset_Ms;
END_IF;

SP_Speed_S := (Base_Speed_X2 * Speed_Ratio_S) + Speed_Offset_S;

IF Core_Dia_T_mm > 0.0 THEN
    SP_Speed_T := ((Base_Speed_X2 * Real_Dia_T_mm) / Core_Dia_T_mm) * Speed_Ratio_T;
ELSE
    SP_Speed_T := Base_Speed_X2 * Speed_Ratio_T;
END_IF;

(* ============================================================================ *)
(* 9.1 BỘ CHUYỂN MẠCH INDEX-REGISTER CHO HMI CHỈNH PID, CALIB VÀ ZERO ĐA TRỤC  *)
(* HMI_Axis_Select (D610): 1=Thu T, 2=Xả X1, 3=Master X2, 4=Ghép Ms, 5=Dầu S, 6=Thắng M, 7=Xả U *)
(* ============================================================================ *)
IF HMI_Axis_Select <= 0 OR HMI_Axis_Select > 7 THEN
    HMI_Axis_Select := 1; (* Mặc định chọn Trục 1: Thu T *)
END_IF;

(* GHI CÀI ĐẶT TỪ HMI VÀO TRỤC ĐANG CHỌN KHI CÓ LỆNH HOẶC THAY ĐỔI *)
IF HMI_Cmd_Save_PID THEN
    CASE HMI_Axis_Select OF
        1: (* Trục Thu T *)
            Kp_T := HMI_Disp_Kp; Ki_T := HMI_Disp_Ki; Kd_T := HMI_Disp_Kd; Calib_Gain_T := HMI_Disp_Calib_Gain; Zero_Offset_T := HMI_Disp_Zero_Offset;
        2: (* Trục Xả X1 *)
            Kp_X1 := HMI_Disp_Kp; Ki_X1 := HMI_Disp_Ki; Kd_X1 := HMI_Disp_Kd; Calib_Gain_X1 := HMI_Disp_Calib_Gain; Zero_Offset_X1 := HMI_Disp_Zero_Offset;
        3: (* Trục Master X2 *)
            Kp_X2 := HMI_Disp_Kp; Ki_X2 := HMI_Disp_Ki; Kd_X2 := HMI_Disp_Kd;
        4: (* Trục Ghép Ms *)
            Kp_Ms := HMI_Disp_Kp; Ki_Ms := HMI_Disp_Ki; Kd_Ms := HMI_Disp_Kd;
        5: (* Trục Dầu S *)
            Kp_S := HMI_Disp_Kp; Ki_S := HMI_Disp_Ki; Kd_S := HMI_Disp_Kd;
        6: (* Trục Thắng M *)
            Kp_M := HMI_Disp_Kp; Ki_M := HMI_Disp_Ki; Kd_M := HMI_Disp_Kd; Calib_Gain_M := HMI_Disp_Calib_Gain; Zero_Offset_M := HMI_Disp_Zero_Offset;
        7: (* Trục Xả U *)
            Kp_U := HMI_Disp_Kp; Ki_U := HMI_Disp_Ki; Kd_U := HMI_Disp_Kd; Calib_Gain_U := HMI_Disp_Calib_Gain; Zero_Offset_U := HMI_Disp_Zero_Offset;
    END_CASE;
    HMI_Cmd_Save_PID := FALSE;
ELSE
    (* ĐỌC THAM SỐ CỦA TRỤC ĐANG CHỌN XUẤT RA Ô HIỂN THỊ TRÊN HMI *)
    CASE HMI_Axis_Select OF
        1: (* Trục Thu T *)
            HMI_Disp_Kp := Kp_T; HMI_Disp_Ki := Ki_T; HMI_Disp_Kd := Kd_T; HMI_Disp_Calib_Gain := Calib_Gain_T; HMI_Disp_Zero_Offset := Zero_Offset_T;
        2: (* Trục Xả X1 *)
            HMI_Disp_Kp := Kp_X1; HMI_Disp_Ki := Ki_X1; HMI_Disp_Kd := Kd_X1; HMI_Disp_Calib_Gain := Calib_Gain_X1; HMI_Disp_Zero_Offset := Zero_Offset_X1;
        3: (* Trục Master X2 *)
            HMI_Disp_Kp := Kp_X2; HMI_Disp_Ki := Ki_X2; HMI_Disp_Kd := Kd_X2; HMI_Disp_Calib_Gain := 1.0; HMI_Disp_Zero_Offset := 0.0;
        4: (* Trục Ghép Ms *)
            HMI_Disp_Kp := Kp_Ms; HMI_Disp_Ki := Ki_Ms; HMI_Disp_Kd := Kd_Ms; HMI_Disp_Calib_Gain := 1.0; HMI_Disp_Zero_Offset := 0.0;
        5: (* Trục Dầu S *)
            HMI_Disp_Kp := Kp_S; HMI_Disp_Ki := Ki_S; HMI_Disp_Kd := Kd_S; HMI_Disp_Calib_Gain := 1.0; HMI_Disp_Zero_Offset := 0.0;
        6: (* Trục Thắng M *)
            HMI_Disp_Kp := Kp_M; HMI_Disp_Ki := Ki_M; HMI_Disp_Kd := Kd_M; HMI_Disp_Calib_Gain := Calib_Gain_M; HMI_Disp_Zero_Offset := Zero_Offset_M;
        7: (* Trục Xả U *)
            HMI_Disp_Kp := Kp_U; HMI_Disp_Ki := Ki_U; HMI_Disp_Kd := Kd_U; HMI_Disp_Calib_Gain := Calib_Gain_U; HMI_Disp_Zero_Offset := Zero_Offset_U;
    END_CASE;
END_IF;

(* XỬ LÝ NÚT BẤM ZERO VÀ CALIB THEO TRỤC ĐANG CHỌN TRÊN HMI *)
IF HMI_Cmd_Zero_Set THEN
    CASE HMI_Axis_Select OF
        1: Zero_Set_T  := TRUE;
        2: Zero_Set_X1 := TRUE;
        6: Zero_Set_M  := TRUE;
        7: Zero_Set_U  := TRUE;
    END_CASE;
    HMI_Cmd_Zero_Set := FALSE;
END_IF;

IF HMI_Cmd_Calib_Set THEN
    CASE HMI_Axis_Select OF
        1: Calib_Set_T  := TRUE;
        2: Calib_Set_X1 := TRUE;
        6: Calib_Set_M  := TRUE;
        7: Calib_Set_U  := TRUE;
    END_CASE;
    HMI_Cmd_Calib_Set := FALSE;
END_IF;

(* TẠO XUNG KÍCH HOẠT PID CHUẨN 10MS TỪ SM409 *)
Trig_PID_10ms := SM409 AND NOT(Prev_SM409);
Prev_SM409 := SM409;

(* 10. GỌI RUN CÁC KHỐI PID THEO NHỊP 10MS (TÍCH HỢP AUTO-TUNING TỰ ĐỘNG) *)
IF Trig_PID_10ms THEN
    (* PID Tốc độ Trục chính Master X2 *)
    pid_X2(
        Enable      := (HMI_PID_Enable AND State_Machine = 1) OR (HMI_Cmd_AutoTune AND HMI_Axis_Select = 3),
        Setpoint    := SP_Speed_X2,
        Feedback    := Feedback_Speed_X2,
        Kp          := Kp_X2, Ki := Ki_X2, Kd := Kd_X2,
        AT_Enable   := (HMI_Cmd_AutoTune AND HMI_Axis_Select = 3)
    );
    PID_Out_X2 := pid_X2.PID_Output;

    (* PID Tốc độ Trục Ghép Ms *)
    pid_Ms(
        Enable      := (HMI_PID_Enable AND State_Machine = 1) OR (HMI_Cmd_AutoTune AND HMI_Axis_Select = 4),
        Setpoint    := SP_Speed_Ms,
        Feedback    := Feedback_Speed_Ms,
        Kp          := Kp_Ms, Ki := Ki_Ms, Kd := Kd_Ms,
        AT_Enable   := (HMI_Cmd_AutoTune AND HMI_Axis_Select = 4)
    );
    PID_Out_Ms := pid_Ms.PID_Output;

    (* PID Tốc độ Trục Tráng Dầu S *)
    pid_S(
        Enable      := (HMI_PID_Enable AND State_Machine = 1) OR (HMI_Cmd_AutoTune AND HMI_Axis_Select = 5),
        Setpoint    := SP_Speed_S,
        Feedback    := Feedback_Speed_S,
        Kp          := Kp_S, Ki := Ki_S, Kd := Kd_S,
        AT_Enable   := (HMI_Cmd_AutoTune AND HMI_Axis_Select = 5)
    );
    PID_Out_S := pid_S.PID_Output;

    (* PID Lực căng Loadcell Trục Kéo Giấy X1 *)
    pid_X1(
        Enable      := (HMI_PID_Enable AND State_Machine = 1) OR (HMI_Cmd_AutoTune AND HMI_Axis_Select = 2),
        Setpoint    := SP_Tension_X1,
        Feedback    := Weight_Net_X1,
        Kp          := Kp_X1, Ki := Ki_X1, Kd := Kd_X1,
        AT_Enable   := (HMI_Cmd_AutoTune AND HMI_Axis_Select = 2)
    );
    PID_Out_X1 := pid_X1.PID_Output;

    (* PID Lực căng Loadcell Cuộn Thu T *)
    pid_T(
        Enable      := (HMI_PID_Enable AND State_Machine = 1) OR (HMI_Cmd_AutoTune AND HMI_Axis_Select = 1),
        Setpoint    := Effective_SP_T,
        Feedback    := Weight_Net_T,
        Kp          := Kp_T, Ki := Ki_T, Kd := Kd_T,
        AT_Enable   := (HMI_Cmd_AutoTune AND HMI_Axis_Select = 1)
    );
    PID_Out_T := pid_T.PID_Output;

    (* PID Lực căng Thắng Từ Xả M *)
    pid_M(
        Enable      := (HMI_PID_Enable AND State_Machine = 1) OR (HMI_Cmd_AutoTune AND HMI_Axis_Select = 6),
        Setpoint    := SP_Tension_M,
        Feedback    := Weight_Net_M,
        Kp          := Kp_M, Ki := Ki_M, Kd := Kd_M,
        AT_Enable   := (HMI_Cmd_AutoTune AND HMI_Axis_Select = 6)
    );
    PID_Out_M := pid_M.PID_Output;

    (* PID Lực căng Trục Xả Metalize U *)
    pid_U(
        Enable      := (HMI_PID_Enable AND State_Machine = 1) OR (HMI_Cmd_AutoTune AND HMI_Axis_Select = 7),
        Setpoint    := SP_Tension_U,
        Feedback    := Weight_Net_U,
        Kp          := Kp_U, Ki := Ki_U, Kd := Kd_U,
        AT_Enable   := (HMI_Cmd_AutoTune AND HMI_Axis_Select = 7)
    );
    PID_Out_U := pid_U.PID_Output;

    (* TỰ ĐỘNG CẬP NHẬT KẾT QUẢ KHI AUTO-TUNE HOÀN THÀNH *)
    IF pid_X2.AT_Done THEN
        Kp_X2 := pid_X2.Tuned_Kp; Ki_X2 := pid_X2.Tuned_Ki; Kd_X2 := pid_X2.Tuned_Kd;
        HMI_Disp_Kp := Kp_X2; HMI_Disp_Ki := Ki_X2; HMI_Disp_Kd := Kd_X2;
    ELSIF pid_Ms.AT_Done THEN
        Kp_Ms := pid_Ms.Tuned_Kp; Ki_Ms := pid_Ms.Tuned_Ki; Kd_Ms := pid_Ms.Tuned_Kd;
        HMI_Disp_Kp := Kp_Ms; HMI_Disp_Ki := Ki_Ms; HMI_Disp_Kd := Kd_Ms;
    ELSIF pid_S.AT_Done THEN
        Kp_S := pid_S.Tuned_Kp; Ki_S := pid_S.Tuned_Ki; Kd_S := pid_S.Tuned_Kd;
        HMI_Disp_Kp := Kp_S; HMI_Disp_Ki := Ki_S; HMI_Disp_Kd := Kd_S;
    ELSIF pid_X1.AT_Done THEN
        Kp_X1 := pid_X1.Tuned_Kp; Ki_X1 := pid_X1.Tuned_Ki; Kd_X1 := pid_X1.Tuned_Kd;
        HMI_Disp_Kp := Kp_X1; HMI_Disp_Ki := Ki_X1; HMI_Disp_Kd := Kd_X1;
    ELSIF pid_T.AT_Done THEN
        Kp_T := pid_T.Tuned_Kp; Ki_T := pid_T.Tuned_Ki; Kd_T := pid_T.Tuned_Kd;
        HMI_Disp_Kp := Kp_T; HMI_Disp_Ki := Ki_T; HMI_Disp_Kd := Kd_T;
    ELSIF pid_M.AT_Done THEN
        Kp_M := pid_M.Tuned_Kp; Ki_M := pid_M.Tuned_Ki; Kd_M := pid_M.Tuned_Kd;
        HMI_Disp_Kp := Kp_M; HMI_Disp_Ki := Ki_M; HMI_Disp_Kd := Kd_M;
    ELSIF pid_U.AT_Done THEN
        Kp_U := pid_U.Tuned_Kp; Ki_U := pid_U.Tuned_Ki; Kd_U := pid_U.Tuned_Kd;
        HMI_Disp_Kp := Kp_U; HMI_Disp_Ki := Ki_U; HMI_Disp_Kd := Kd_U;
    END_IF;

    (* TẮT CỜ AUTO-TUNE DUY NHẤT TẠI 1 ĐIỂM CHỐNG CẢNH BÁO DOUBLE-COIL C9300 *)
    IF pid_X2.AT_Done OR pid_Ms.AT_Done OR pid_S.AT_Done OR pid_X1.AT_Done OR pid_T.AT_Done OR pid_M.AT_Done OR pid_U.AT_Done THEN
        HMI_Cmd_AutoTune   := FALSE;
        HMI_Status_AT_Done := TRUE;
    END_IF;
    
    (* Cập nhật cờ báo bận Auto-Tune *)
    HMI_Status_AT_Busy := pid_T.AT_Busy OR pid_X1.AT_Busy OR pid_X2.AT_Busy OR pid_Ms.AT_Busy OR pid_S.AT_Busy OR pid_M.AT_Busy OR pid_U.AT_Busy;
END_IF;

(* 11. TÍNH TOÁN XUẤT ÁP TỐC ĐỘ VÀ TORQUE CHO TỪNG TRỤC (FLOAT) *)
IF State_Machine = 0 THEN
    (* KHI MÁY DỪNG: KIỂM TRA CHẾ ĐỘ TEST RIÊNG BIỆT TỪNG TRỤC HOẶC BÒ CHẬM RỬA MÁY *)
    IF HMI_Test_X2 THEN Calc_Speed_X2 := Test_Speed_X2; ELSE Calc_Speed_X2 := 0.0; END_IF;
    IF HMI_Test_X1 THEN Calc_Speed_X1 := Test_Speed_X1; ELSE Calc_Speed_X1 := 0.0; END_IF;

    IF HMI_Test_Ms THEN
        Calc_Speed_Ms := Test_Speed_Ms;
    ELSIF Anti_Dry_Rotate_Ms AND Max_Speed_MPM > 0.0 THEN
        Calc_Speed_Ms := (Anti_Dry_Crawl_Speed * 16000.0) / Max_Speed_MPM;
    ELSE
        Calc_Speed_Ms := 0.0;
    END_IF;

    IF HMI_Test_S THEN
        Calc_Speed_S := Test_Speed_S;
    ELSIF Anti_Dry_Rotate_S AND Max_Speed_MPM > 0.0 THEN
        Calc_Speed_S := (Anti_Dry_Crawl_Speed * 16000.0) / Max_Speed_MPM;
    ELSE
        Calc_Speed_S := 0.0;
    END_IF;

    IF HMI_Test_T THEN
        Calc_Speed_T  := Test_Speed_T;
        Calc_Torque_T := Test_Torque_T;
    ELSE
        Calc_Speed_T  := 0.0;
        Calc_Torque_T := 0.0;
    END_IF;

    IF HMI_Test_M THEN
        Calc_Torque_M := Test_Torque_M;
    ELSIF Hold_Torque_Stop_M THEN
        Calc_Torque_M := (Base_Torque_M * 160.0);
    ELSE
        Calc_Torque_M := 0.0;
    END_IF;

    IF HMI_Test_U THEN
        Calc_Speed_U := Test_Speed_U;
    ELSIF Hold_Torque_Stop_U THEN
        Calc_Speed_U := (Init_Holding_Torque_U * 160.0);
    ELSE
        Calc_Speed_U := 0.0;
    END_IF;

ELSE
    (* KHI MÁY CHẠY TỰ ĐỘNG *)
    Calc_Speed_X2 := SP_Speed_X2 + PID_Out_X2;
    Calc_Speed_X1 := SP_Speed_X1 + PID_Out_X1;
    Calc_Speed_Ms := SP_Speed_Ms + PID_Out_Ms;
    Calc_Speed_S  := SP_Speed_S  + PID_Out_S;
    Calc_Speed_T  := SP_Speed_T;
    Calc_Torque_T := (Effective_SP_T * 160.0) + PID_Out_T;

    IF Real_Dia_U_mm > 0.0 THEN
        Calc_Speed_U := ((Calc_Speed_X2 * Max_Dia_U_mm) / Real_Dia_U_mm) + PID_Out_U;
    ELSE
        Calc_Speed_U := Calc_Speed_X2 + PID_Out_U;
    END_IF;

    (* 3 Pha Torque Thắng M (0..100% quy đổi ra 0..16000) *)
    IF Rev_Count_M <= 5 THEN
        Base_Torque_M := Init_Holding_Torque_M;
    ELSIF (Max_Dia_M_mm - Core_Dia_M_mm) > 0.0 THEN
        Base_Torque_M := Min_Torque_M + (((Max_Torque_M - Min_Torque_M) * (Real_Dia_M_mm - Core_Dia_M_mm)) / (Max_Dia_M_mm - Core_Dia_M_mm));
    ELSE
        Base_Torque_M := Min_Torque_M;
    END_IF;
    Calc_Torque_M := (Base_Torque_M * 160.0) + PID_Out_M;
END_IF;

(* KHỐNG CHẾ BIÊN AN TOÀN 0..16000 CHO TOÀN BỘ 8 KÊNH DAC (HIGH RESOLUTION) *)
IF Calc_Speed_T  < 0.0 THEN Calc_Speed_T  := 0.0; ELSIF Calc_Speed_T  > 16000.0 THEN Calc_Speed_T  := 16000.0; END_IF;
IF Calc_Torque_T < 0.0 THEN Calc_Torque_T := 0.0; ELSIF Calc_Torque_T > 16000.0 THEN Calc_Torque_T := 16000.0; END_IF;
IF Calc_Speed_X1 < 0.0 THEN Calc_Speed_X1 := 0.0; ELSIF Calc_Speed_X1 > 16000.0 THEN Calc_Speed_X1 := 16000.0; END_IF;
IF Calc_Speed_X2 < 0.0 THEN Calc_Speed_X2 := 0.0; ELSIF Calc_Speed_X2 > 16000.0 THEN Calc_Speed_X2 := 16000.0; END_IF;
IF Calc_Speed_Ms < 0.0 THEN Calc_Speed_Ms := 0.0; ELSIF Calc_Speed_Ms > 16000.0 THEN Calc_Speed_Ms := 16000.0; END_IF;
IF Calc_Torque_M < 0.0 THEN Calc_Torque_M := 0.0; ELSIF Calc_Torque_M > 16000.0 THEN Calc_Torque_M := 16000.0; END_IF;
IF Calc_Speed_S  < 0.0 THEN Calc_Speed_S  := 0.0; ELSIF Calc_Speed_S  > 16000.0 THEN Calc_Speed_S  := 16000.0; END_IF;
IF Calc_Speed_U  < 0.0 THEN Calc_Speed_U  := 0.0; ELSIF Calc_Speed_U  > 16000.0 THEN Calc_Speed_U  := 16000.0; END_IF;

(* 12. THỰC THI FB CC-LINK XUẤT ÁP 8 KÊNH DAC (TRUYỀN TRỰC TIẾP BIẾN FLOAT) *)
fbCCLink(
    Enable          := TRUE,
    ResetErr        := HMI_Reset_Error,
    Auto_Mode       := HMI_Auto_Mode,
    Set_Speed_T     := Calc_Speed_T,
    Set_Torque_T    := Calc_Torque_T,
    Set_Speed_X1    := Calc_Speed_X1,
    Set_Speed_X2    := Calc_Speed_X2,
    Set_Speed_Ms    := Calc_Speed_Ms,
    Set_Torque_M    := Calc_Torque_M,
    Set_Speed_S     := Calc_Speed_S,
    Set_Speed_U     := Calc_Speed_U
);

(* 13. TỰ ĐỘNG BÁO GIẢM TỐC VÀ DỪNG MÁY KHI ĐẠT CHIỀU DÀI MÉT CÀI ĐẶT *)
IF Set_Target_Length > 0.0 AND State_Machine = 1 THEN
    (* Pha 1: Giảm tốc về Min_Speed khi còn cách đích khoảng cách Decel_Distance_Meters *)
    IF Decel_Distance_Meters > 0.0 AND Total_Length_Meters >= (Set_Target_Length - Decel_Distance_Meters) THEN
        Auto_Decel_Flag := TRUE;
        IF Target_Line_MPM > Min_Speed_MPM THEN Target_Line_MPM := Min_Speed_MPM; END_IF;
    ELSE
        Auto_Decel_Flag := FALSE;
    END_IF;

    (* Pha 2: Dừng máy hoàn toàn khi đã đủ tổng mét màng cài đặt *)
    IF Total_Length_Meters >= Set_Target_Length THEN
        State_Machine    := 0;
        Target_Line_MPM  := 0.0;
        Current_Line_MPM := 0.0;
        Auto_Decel_Flag  := FALSE;
    END_IF;
END_IF;

(* 14. CẬP NHẬT MÃ TRẠNG THÁI HIỂN THỊ TIẾNG VIỆT TRÊN HMI CHO CÔNG NHÂN *)
(* 0: Sẵn sàng | 1: Báo lỗi Servo | 2: Đang chạy Auto | 3: Đang bò nối màng | 4: Hoàn thành đơn hàng *)
IF Servo_Not_Ready_Fault THEN
    HMI_Status_Text_Code := 1; (* Báo lỗi 5 Servo *)
ELSIF State_Machine = 1 THEN
    HMI_Status_Text_Code := 2; (* Đang chạy tự động *)
ELSIF Cmd_Jog_Crawl THEN
    HMI_Status_Text_Code := 3; (* Đang bò chậm nối màng *)
ELSIF Auto_Decel_Flag OR (Set_Target_Length > 0.0 AND Total_Length_Meters >= Set_Target_Length) THEN
    HMI_Status_Text_Code := 4; (* Đã hoàn thành đơn hàng *)
ELSE
    HMI_Status_Text_Code := 0; (* Máy dừng - Sẵn sàng chạy *)
END_IF;
END_PROGRAM

FUNCTION_BLOCK FFB_CCLINK_CONTROL
VAR_INPUT
  Enable : BOOL;  (* Cho phep FB hoat dong *)
  ResetErr : BOOL;  (* Nut reset loi he thong *)
  Auto_Mode : BOOL;  (* Che do Auto / Manual *)
  Set_Speed_T : REAL;  (* CH1 Speed Thu T (0.0..16000.0) *)
  Set_Torque_T : REAL;  (* CH2 Torque Thu T (0.0..16000.0) *)
  Set_Speed_X1 : REAL;  (* CH3 Speed Xa X1 (0.0..16000.0) *)
  Set_Speed_X2 : REAL;  (* CH4 Speed Master X2 (0.0..16000.0) *)
  Set_Speed_Ms : REAL;  (* CH5 Speed Ghep Ms (0.0..16000.0) *)
  Set_Torque_M : REAL;  (* CH6 Torque Thang M (0.0..16000.0) *)
  Set_Speed_S : REAL;  (* CH7 Speed Trang Dau S (0.0..16000.0) *)
  Set_Speed_U : REAL;  (* CH8 Speed Xa U (0.0..16000.0) *)
  DO_Y8_Cmd : BOOL;  (* Lenh ngo ra Y8 St 5 (M1336) *)
  DO_Y9_Cmd : BOOL;  (* Lenh ngo ra Y9 St 5 (M1337) *)
END_VAR
VAR_OUTPUT
  CCLink_OK : BOOL;  (* Trang thai mang CC-Link OK *)
  HasError : BOOL;  (* Bao loi tong truyen thong module *)
  ADC_CH1_Val : REAL;  (* Gia tri thuc ADC CH1 (REAL) *)
  ADC_CH2_Val : REAL;  (* Gia tri thuc ADC CH2 (REAL) *)
  ADC_CH3_Val : REAL;  (* Gia tri thuc ADC CH3 (REAL) *)
  ADC_CH4_Val : REAL;  (* Gia tri thuc ADC CH4 (REAL) *)
  ADC_CH5_Val : REAL;  (* Gia tri thuc ADC CH5 (REAL) *)
  ADC_CH6_Val : REAL;  (* Gia tri thuc ADC CH6 (REAL) *)
  ADC_CH7_Val : REAL;  (* Gia tri thuc ADC CH7 (REAL) *)
  ADC_CH8_Val : REAL;  (* Gia tri thuc ADC CH8 (REAL) *)
  ADC_CH1_Raw : WORD;  (* Gia tri tho D500 ADC CH1 *)
  ADC_CH2_Raw : WORD;  (* Gia tri tho D501 ADC CH2 *)
  ADC_CH3_Raw : WORD;  (* Gia tri tho D502 ADC CH3 *)
  ADC_CH4_Raw : WORD;  (* Gia tri tho D503 ADC CH4 *)
  ADC_CH5_Raw : WORD;  (* Gia tri tho D504 ADC CH5 *)
  ADC_CH6_Raw : WORD;  (* Gia tri tho D505 ADC CH6 *)
  ADC_CH7_Raw : WORD;  (* Gia tri tho D506 ADC CH7 *)
  ADC_CH8_Raw : WORD;  (* Gia tri tho D507 ADC CH8 *)
  DI_X0_State : BOOL;  (* Trang thai ngo vao X0 St 5 (M1136) *)
  DI_X1_State : BOOL;  (* Trang thai ngo vao X1 St 5 (M1137) *)
END_VAR
(* ============================================================================ *)
(* FUNCTION BLOCK BODY: FB_CCLINK_CONTROL (CHUẨN CHÍNH THỨC MANUAL MITSUBISHI)  *)
(* TRẠM 1: ADC INPUT  (AJ65VBTCU-68ADV  - D500..D507 | RWw0: D520 = 16#00FF)    *)
(* TRẠM 2: DAC OUTPUT (AJ65VBTCU-68DAVN - D524..D535 | XUẤT 5.0V D524)          *)
(* TRẠM 3: DIGITAL IO (AJ65SBTB1-16DT   - RX: M1072..M1079 | RY: M1272..M1279) *)
(* ============================================================================ *)

IF Enable THEN

    (* 1. TRẠNG THÁI MẠNG *)
    CCLink_OK := (NOT SB0020) AND (NOT SB0049);
    HasError  := SB0020 OR SB0049;

    (* 2. CẤU HÌNH BẮT BUỘC THEO MANUAL MITSUBISHI CHO AJ65VBTCU-68ADV *)
    (* RWw0 (D520): Cho phép chuyển đổi A/D cả 8 kênh (16#00FF = 255) *)
    D520 := 16#00FF; 
    (* RWw1 (D521): Dải ngõ vào 0..10V cho cả 8 kênh *)
    D521 := 16#0000; 

    (* Tự động gửi xung bắt tay RY19 (M1225) nạp thông số vào module *)
    IF M1032 THEN 
        M1225 := TRUE;  (* Bật xung nạp tham số *)
    ELSE 
        M1225 := FALSE; (* Tự ngắt khi nạp xong -> Đèn RUN sáng đứng *)
    END_IF;

    (* Bật cờ chuyển đổi RY0..RY7 *)
    M1200 := CCLink_OK; M1201 := CCLink_OK; M1202 := CCLink_OK; M1203 := CCLink_OK;
    M1204 := CCLink_OK; M1205 := CCLink_OK; M1206 := CCLink_OK; M1207 := CCLink_OK;

    (* 3. BẬT CỜ XUẤT ÁP CHO TRẠM 2 DAC *)
    M1232 := CCLink_OK; M1233 := CCLink_OK; M1234 := CCLink_OK; M1235 := CCLink_OK;

    (* 4. ĐỌC 8 KÊNH ANALOG INPUT TỪ TRẠM 1 ADC (D500..D507) *)
    ADC_CH1_Raw := D500;
    ADC_CH2_Raw := D501;
    ADC_CH3_Raw := D502;
    ADC_CH4_Raw := D503;
    ADC_CH5_Raw := D504;
    ADC_CH6_Raw := D505;
    ADC_CH7_Raw := D506;
    ADC_CH8_Raw := D507;

    (* Chuyển đổi sang số thực REAL *)
    ADC_CH1_Val := INT_TO_REAL(WORD_TO_INT(D500));
    ADC_CH2_Val := INT_TO_REAL(WORD_TO_INT(D501));
    ADC_CH3_Val := INT_TO_REAL(WORD_TO_INT(D502));
    ADC_CH4_Val := INT_TO_REAL(WORD_TO_INT(D503));
    ADC_CH5_Val := INT_TO_REAL(WORD_TO_INT(D504));
    ADC_CH6_Val := INT_TO_REAL(WORD_TO_INT(D505));
    ADC_CH7_Val := INT_TO_REAL(WORD_TO_INT(D506));
    ADC_CH8_Val := INT_TO_REAL(WORD_TO_INT(D507));

    (* 5. XUẤT ÁP 5.0V RA DAC TRẠM 2 (D524 / D528) *)
    D524 := INT_TO_WORD(2000);  (* Xuất 5.0V Kênh 1 *)
    D528 := INT_TO_WORD(2000);

    (* CH2..CH4 *)
    IF Set_Torque_T < 0.0 THEN D525 := INT_TO_WORD(0); ELSIF Set_Torque_T > 4000.0 THEN D525 := INT_TO_WORD(4000); ELSE D525 := INT_TO_WORD(REAL_TO_INT(Set_Torque_T)); END_IF;
    IF Set_Speed_X1 < 0.0 THEN D526 := INT_TO_WORD(0); ELSIF Set_Speed_X1 > 4000.0 THEN D526 := INT_TO_WORD(4000); ELSE D526 := INT_TO_WORD(REAL_TO_INT(Set_Speed_X1)); END_IF;
    IF Set_Speed_X2 < 0.0 THEN D527 := INT_TO_WORD(0); ELSIF Set_Speed_X2 > 4000.0 THEN D527 := INT_TO_WORD(4000); ELSE D527 := INT_TO_WORD(REAL_TO_INT(Set_Speed_X2)); END_IF;

    (* 6. XỬ LÝ DIGITAL REMOTE I/O TRẠM 3 (AJ65SBTB1-16DT: RX: M1072..M1076 | RY: M1272..M1273) *)
    DI_X0_State := M1072;
    DI_X1_State := M1073;
    M1272 := DO_Y8_Cmd;
    M1273 := DO_Y9_Cmd;

    (* 7. RESET LỖI *)
    M1226 := ResetErr OR M1111;
    M1258 := ResetErr OR M1111;

END_IF;
END_FUNCTION_BLOCK

FUNCTION_BLOCK FB_TENSION_PID
VAR_INPUT
  Enable : BOOL;  (* Cho phep PID hoat dong *)
  Reset : BOOL;  (* Reset tich luy I *)
  Setpoint : REAL;  (* Gia tri luc cang/toc do cai dat (REAL) *)
  Feedback : REAL;  (* Gia tri phan hoi tu Loadcell/Encoder (REAL) *)
  Kp : REAL;  (* He so Kp (REAL) *)
  Ki : REAL;  (* He so Ki (REAL) *)
  Kd : REAL;  (* He so Kd (REAL) *)
  Deadband : REAL;  (* Vung chet khong chinh (REAL) *)
  Out_Min : REAL;  (* Gioi han dau ra toi thieu (REAL) *)
  Out_Max : REAL;  (* Gioi han dau ra toi da (REAL) *)
  AT_Enable : BOOL;  (* Lenh kich hoat Auto-Tuning tu dong do tim Kp, Ki, Kd *)
  AT_Step : REAL;  (* Bien do xung buoc nhay test Auto-Tune (vi du 200.0..400.0) *)
END_VAR
VAR_OUTPUT
  PID_Output : REAL;  (* Gia tri bu toc do torque cho DAC (REAL) *)
  Error : REAL;  (* Do lech e(k) (REAL) *)
  AT_Done : BOOL;  (* Co bao da Auto-Tuning xong *)
  AT_Busy : BOOL;  (* Co bao dang trong qua trinh Auto-Tuning *)
  Tuned_Kp : REAL;  (* He so Kp vua do tim duoc *)
  Tuned_Ki : REAL;  (* He so Ki vua do tim duoc *)
  Tuned_Kd : REAL;  (* He so Kd vua do tim duoc *)
END_VAR
VAR
  Error_Prev : REAL;  (* Do lech vong truoc (REAL) *)
  I_Term : REAL;  (* Thanh phan Tich phan I (REAL) *)
  P_Term : REAL;  (* Thanh phan Ty le P (REAL) *)
  D_Term : REAL;  (* Thanh phan Dao ham D (REAL) *)
  AT_State : INT;  (* Trang thai State Machine cua Auto-Tune *)
  AT_Cycle_Count : INT;  (* Dem so chu ky dao dong Limit Cycle *)
  AT_Timer_10ms : DINT;  (* Timer do chu ky dao dong (nhip 10ms) *)
  AT_Period_Tu : REAL;  (* Chu ky dao dong rieng Tu (giay) *)
  AT_Ku : REAL;  (* Do khuech dai gioi han Ku *)
  AT_PV_Max : REAL;  (* Gia tri Feedback dinh cao nhat *)
  AT_PV_Min : REAL;  (* Gia tri Feedback day thap nhat *)
  AT_Base_Out : REAL;  (* Muc dau ra co ban truoc khi test *)
  AT_Relay_State : BOOL;  (* Trang thai Relay Output (+Step / -Step) *)
  Test_Step : REAL;  (* Bien do buoc nhay test noi bo *)
END_VAR
(* ============================================================================ *)
(* FUNCTION BLOCK: FB_TENSION_PID (ĐIỀU KHIỂN PID & AUTO-TUNING TỰ ĐỘNG TÌM THÔNG SỐ) *)
(* PHƯƠNG PHÁP AUTO-TUNING: RELAY FEEDBACK LIMIT-CYCLE (ZIEGLER-NICHOLS CẢI TIẾN) *)
(* ============================================================================ *)

IF NOT Enable THEN
    PID_Output := 0.0;
    I_Term     := 0.0;
    Error_Prev := 0.0;
    AT_Busy    := FALSE;
    AT_State   := 0;
    RETURN;
END_IF;

IF Reset THEN
    I_Term     := 0.0;
    Error_Prev := 0.0;
    PID_Output := 0.0;
    AT_Busy    := FALSE;
    AT_State   := 0;
    AT_Done    := FALSE;
    RETURN;
END_IF;

(* ============================================================================ *)
(* 1. CHẾ ĐỘ AUTO-TUNING (DÒ THÔNG SỐ TỰ ĐỘNG BẰNG RELAY LIMIT-CYCLE)           *)
(* ============================================================================ *)
IF AT_Enable THEN
    AT_Busy := TRUE;
    AT_Done := FALSE;
    
    (* Sử dụng biến nội bộ Test_Step để không ghi đè vào VAR_INPUT AT_Step *)
    IF AT_Step > 0.0 THEN
        Test_Step := AT_Step;
    ELSE
        Test_Step := 200.0; (* Mặc định 200 đơn vị DAC ~ 5% *)
    END_IF;

    CASE AT_State OF
        0: (* KHỞI TẠO BƯỚC TEST *)
            AT_Base_Out     := PID_Output;
            AT_PV_Max       := Feedback;
            AT_PV_Min       := Feedback;
            AT_Cycle_Count  := 0;
            AT_Timer_10ms   := 0;
            AT_Relay_State  := TRUE;
            AT_State        := 1;

        1: (* THỰC THI DAO ĐỘNG BẬT/TẮT RELAY QUA SETPOINT *)
            AT_Timer_10ms := AT_Timer_10ms + 1;

            (* Theo dõi giá trị đỉnh/đáy của Feedback *)
            IF Feedback > AT_PV_Max THEN AT_PV_Max := Feedback; END_IF;
            IF Feedback < AT_PV_Min THEN AT_PV_Min := Feedback; END_IF;

            (* Điều khiển Relay đảo trạng thái khi vượt qua Setpoint *)
            IF AT_Relay_State THEN
                PID_Output := AT_Base_Out + Test_Step;
                IF Feedback >= Setpoint THEN
                    AT_Relay_State := FALSE;
                END_IF;
            ELSE
                PID_Output := AT_Base_Out - Test_Step;
                IF Feedback < Setpoint THEN
                    AT_Relay_State := TRUE;
                    AT_Cycle_Count := AT_Cycle_Count + 1; (* Đếm xong 1 chu kỳ hoàn chỉnh *)
                END_IF;
            END_IF;

            (* Khi hoàn thành đủ 3 chu kỳ dao động chuẩn *)
            IF AT_Cycle_Count >= 3 THEN
                AT_State := 2;
            END_IF;

        2: (* TÍNH TOÁN BỘ THÔNG SỐ TUNED_KP, TUNED_KI, TUNED_KD *)
            (* Chu kỳ dao động riêng Tu (giây) = tổng thời gian 3 chu kỳ / 3 *)
            IF AT_Timer_10ms > 0 THEN
                AT_Period_Tu := (DINT_TO_REAL(AT_Timer_10ms) * 0.01) / 3.0;
            ELSE
                AT_Period_Tu := 1.0;
            END_IF;

            (* Biên độ dao động đáp ứng A = (PV_Max - PV_Min) / 2 *)
            IF (AT_PV_Max - AT_PV_Min) > 0.1 THEN
                (* Độ khuếch đại tới hạn Ku = 4 * Test_Step / (PI * A) *)
                AT_Ku := (4.0 * Test_Step) / (3.141593 * ((AT_PV_Max - AT_PV_Min) / 2.0));
            ELSE
                AT_Ku := 1.0;
            END_IF;

            (* TÍNH THEO CÔNG THỨC ZIEGLER-NICHOLS CHỐNG VỌT LỐ (NO-OVERSHOOT) *)
            Tuned_Kp := AT_Ku * 0.35;                   (* Kp an toàn êm ái *)
            
            IF AT_Period_Tu > 0.05 THEN
                Tuned_Ki := Tuned_Kp * (0.01 / (AT_Period_Tu * 0.85)); (* Ki cho chu kỳ 10ms *)
                Tuned_Kd := Tuned_Kp * ((AT_Period_Tu * 0.12) / 0.01); (* Kd cho chu kỳ 10ms *)
            ELSE
                Tuned_Ki := Tuned_Kp * 0.05;
                Tuned_Kd := Tuned_Kp * 0.02;
            END_IF;

            (* Khống chế biên an toàn *)
            IF Tuned_Kp < 0.1 THEN Tuned_Kp := 0.1; ELSIF Tuned_Kp > 20.0 THEN Tuned_Kp := 20.0; END_IF;
            IF Tuned_Ki < 0.001 THEN Tuned_Ki := 0.001; ELSIF Tuned_Ki > 5.0 THEN Tuned_Ki := 5.0; END_IF;
            IF Tuned_Kd < 0.0 THEN Tuned_Kd := 0.0; ELSIF Tuned_Kd > 5.0 THEN Tuned_Kd := 5.0; END_IF;

            AT_Busy  := FALSE;
            AT_Done  := TRUE;
            AT_State := 0;
    END_CASE;

    (* Giới hạn biên đầu ra trong lúc test *)
    IF PID_Output > Out_Max THEN PID_Output := Out_Max; END_IF;
    IF PID_Output < Out_Min THEN PID_Output := Out_Min; END_IF;
    RETURN;
END_IF;

(* Khi tắt AT_Enable *)
IF AT_Busy THEN
    AT_Busy  := FALSE;
    AT_State := 0;
END_IF;

(* ============================================================================ *)
(* 2. CHẾ ĐỘ ĐIỀU KHIỂN PID TIÊU CHUẨN (NORMAL RUNNING)                        *)
(* ============================================================================ *)

(* 1. TÍNH ĐỘ LỆCH ERROR E(K) *)
Error := Setpoint - Feedback;

(* 2. BỘ LỌC VÙNG CHẾT DEADBAND *)
IF ABS(Error) <= Deadband THEN
    Error := 0.0;
END_IF;

(* 3. TÍNH THÀNH PHẦN PROPORTIONAL (P) *)
P_Term := Error * Kp;

(* 4. TÍNH THÀNH PHẦN INTEGRAL (I) VỚI CHỐNG BÃO HÒA ANTI-WINDUP *)
I_Term := I_Term + (Error * Ki);

IF Out_Max > Out_Min THEN
    IF I_Term > Out_Max THEN
        I_Term := Out_Max;
    ELSIF I_Term < Out_Min THEN
        I_Term := Out_Min;
    END_IF;
END_IF;

(* 5. TÍNH THÀNH PHẦN DERIVATIVE (D) *)
D_Term := (Error - Error_Prev) * Kd;
Error_Prev := Error;

(* 6. TỔNG HỢP NỔI PID VÀ ÉP BIÊN OUT_MIN..OUT_MAX *)
PID_Output := P_Term + I_Term + D_Term;

IF Out_Max > Out_Min THEN
    IF PID_Output > Out_Max THEN
        PID_Output := Out_Max;
    ELSIF PID_Output < Out_Min THEN
        PID_Output := Out_Min;
    END_IF;
END_IF;
END_FUNCTION_BLOCK

PROGRAM POU_INIT
(* ============================================================================ *)
(* TÊN CHƯƠNG TRÌNH : INIT_PROGRAM (INITIAL EXECUTION POU - KHỞI TẠO HỆ THỐNG)    *)
(* HỆ THỐNG        : MÁY GHÉP MÀNG METALIZE TỰ ĐỘNG - MITSUBISHI Q02U PLC       *)
(* KIỂU DỮ LIỆU    : SỐ THỰC FLOAT / REAL (CHUẨN IEC)                          *)
(* MỤC ĐÍCH        : KHỞI TẠO TỶ SỐ TRUYỀN, ĐƯỜNG KÍNH LÔ, THÔNG SỐ TỐC ĐỘ,     *)
(*                   LỰC CĂNG, PID VÀ BẢO VỆ CHỐNG LỖI CHIA CHO 0 (ZERO DIV)    *)
(* GHI CHÚ QUAN TRỌNG: POU này đã được cài đặt là "Initial" trong PLC Parameter  *)
(*                   nên CPU chỉ quét đúng 1 lần khi chuyển sang RUN (Không     *)
(*                   cần dùng tiếp cờ SM402).                                   *)
(* ============================================================================ *)

(* ---------------------------------------------------------------------------- *)
(* 1. KHỞI TẠO TỐC ĐỘ TỐI ĐA MOTOR (RPM - REAL)                                *)
(* ---------------------------------------------------------------------------- *)
IF Max_RPM_X2 <= 0.0 THEN Max_RPM_X2 := 1000.0; END_IF; (* Trục Master X2: Max 1000 RPM *)
IF Max_RPM_X1 <= 0.0 THEN Max_RPM_X1 := 1000.0; END_IF; (* Trục Kéo X1:    Max 1000 RPM *)
IF Max_RPM_Ms <= 0.0 THEN Max_RPM_Ms := 3000.0; END_IF; (* Trục Ghép Ms:   Max 3000 RPM *)
IF Max_RPM_S  <= 0.0 THEN Max_RPM_S  := 3000.0; END_IF; (* Trục Dầu S:     Max 3000 RPM *)
IF Max_RPM_T  <= 0.0 THEN Max_RPM_T  := 1500.0; END_IF; (* Trục Thu T:     Max 1500 RPM *)

(* ---------------------------------------------------------------------------- *)
(* 2. KHỞI TẠO TỶ SỐ TRUYỀN HỘP SỐ THỰC TẾ (GEAR RATIO - REAL)                *)
(* ---------------------------------------------------------------------------- *)
IF Gear_Ratio_T  <= 0.0 THEN Gear_Ratio_T  := 10.1; END_IF; (* Thu T:     10.1 : 1 (D620) *)
IF Gear_Ratio_X1 <= 0.0 THEN Gear_Ratio_X1 := 8.0;  END_IF; (* Xả X1:     8.0  : 1 (D622) *)
IF Gear_Ratio_X2 <= 0.0 THEN Gear_Ratio_X2 := 8.0;  END_IF; (* Master X2: 8.0  : 1 (D624) *)
IF Gear_Ratio_Ms <= 0.0 THEN Gear_Ratio_Ms := 10.0; END_IF; (* Ghép Ms:   10.0 : 1 (D626) *)
IF Gear_Ratio_S  <= 0.0 THEN Gear_Ratio_S  := 10.0; END_IF; (* Dầu S:     10.0 : 1 (D628) *)
IF Gear_Ratio_U  <= 0.0 THEN Gear_Ratio_U  := 1.0;  END_IF; (* Xả U:      1.0  : 1 (D630) *)

(* ---------------------------------------------------------------------------- *)
(* 3. KHỞI TẠO ĐƯỜNG KÍNH LÔ CƠ CẤU (ROLLER DIAMETER - mm - REAL)              *)
(* ---------------------------------------------------------------------------- *)
IF Dia_X1_Roller_mm <= 0.0 THEN Dia_X1_Roller_mm := 300.5; END_IF; (* Lô Kéo X1:    300.5 mm (D638) *)
IF Dia_X2_Roller_mm <= 0.0 THEN Dia_X2_Roller_mm := 300.5; END_IF; (* Lô Master X2: 300.5 mm (D642) *)
IF Dia_Ms_Roller_mm <= 0.0 THEN Dia_Ms_Roller_mm := 200.0; END_IF; (* Lô Ghép Ms:   200.0 mm (D640) *)
IF Dia_S_Roller_mm  <= 0.0 THEN Dia_S_Roller_mm  := 100.0; END_IF; (* Lô Dầu S:     100.0 mm (D648) *)

(* ---------------------------------------------------------------------------- *)
(* 4. KHỞI TẠO ĐƯỜNG KÍNH LÕI (CORE) VÀ ĐƯỜNG KÍNH MAX (MAX DIA) (mm - REAL)    *)
(* ---------------------------------------------------------------------------- *)
IF Core_Dia_T_mm <= 0.0 THEN Core_Dia_T_mm := 76.0;   END_IF; (* Lõi cuộn Thu T:  76.0 mm (D644) *)
IF Core_Dia_M_mm <= 0.0 THEN Core_Dia_M_mm := 76.0;   END_IF; (* Lõi cuộn Xả M:   76.0 mm (D645) *)
IF Core_Dia_U_mm <= 0.0 THEN Core_Dia_U_mm := 76.0;   END_IF; (* Lõi cuộn Xả U:   76.0 mm (D647) *)

IF Max_Dia_T_mm  <= 0.0 THEN Max_Dia_T_mm  := 1000.0; END_IF; (* Cuộn Thu T max: 1000.0 mm (D646) *)
IF Max_Dia_M_mm  <= 0.0 THEN Max_Dia_M_mm  := 600.0;  END_IF; (* Cuộn Xả M max:   600.0 mm (D649) *)
IF Max_Dia_U_mm  <= 0.0 THEN Max_Dia_U_mm  := 800.0;  END_IF; (* Cuộn Xả U max:   800.0 mm (D650) *)

(* ---------------------------------------------------------------------------- *)
(* 5. KHỞI TẠO ĐƯỜNG KÍNH BAN ĐẦU KHI MỚI BẬT NGUỒN (REAL)                     *)
(* ---------------------------------------------------------------------------- *)
(* Cuộn Thu T bắt đầu từ Lõi *)
IF Real_Dia_T_mm < Core_Dia_T_mm OR Real_Dia_T_mm > Max_Dia_T_mm THEN
    Real_Dia_T_mm := Core_Dia_T_mm; (* 76.0 mm - D724 *)
END_IF;

(* Cuộn Xả M & U bắt đầu từ cuộn đầy *)
IF Real_Dia_M_mm < Core_Dia_M_mm OR Real_Dia_M_mm > Max_Dia_M_mm THEN
    Real_Dia_M_mm := Max_Dia_M_mm;  (* 600.0 mm - D722 *)
END_IF;

IF Real_Dia_U_mm < Core_Dia_U_mm OR Real_Dia_U_mm > Max_Dia_U_mm THEN
    Real_Dia_U_mm := Max_Dia_U_mm;  (* 800.0 mm - D720 *)
END_IF;

(* ---------------------------------------------------------------------------- *)
(* 6. KHỞI TẠO TỶ LỆ TỐC ĐỘ VÀ BÙ TỐC (SPEED RATIO - REAL, 1.0 = 100%)         *)
(* ---------------------------------------------------------------------------- *)
IF Speed_Ratio_T  <= 0.0 THEN Speed_Ratio_T  := 1.05; END_IF; (* Chạy nhanh hơn 5% giữ căng (D756) *)
IF Speed_Ratio_X1 <= 0.0 THEN Speed_Ratio_X1 := 1.00; END_IF; (* Đồng bộ 100.0% (D758) *)
IF Speed_Ratio_Ms <= 0.0 THEN Speed_Ratio_Ms := 1.00; END_IF; (* Đồng bộ 100.0% (D762) *)
IF Speed_Ratio_S  <= 0.0 THEN Speed_Ratio_S  := 1.00; END_IF; (* Đồng bộ 100.0% (D766) *)

(* ---------------------------------------------------------------------------- *)
(* 7. KHỞI TẠO GIỚI HẠN TỐC ĐỘ DÂY CHUYỀN (m/phút - REAL)                      *)
(* ---------------------------------------------------------------------------- *)
IF Max_Speed_MPM         <= 0.0 THEN Max_Speed_MPM         := 100.0; END_IF; (* Max 100.0 m/p (D602) *)
IF Min_Speed_MPM         <= 0.0 THEN Min_Speed_MPM         := 2.0;   END_IF; (* Min 2.0 m/p (D603) *)
IF Release_Pen_Speed_MPM <= 0.0 THEN Release_Pen_Speed_MPM := 2.0;   END_IF; (* Tốc độ nhả pen (D604) *)
IF Ramp_Accel_Rate       <= 0.0 THEN Ramp_Accel_Rate       := 0.5;   END_IF; (* Gia tốc tăng tốc (D606) *)
IF Ramp_Decel_Rate       <= 0.0 THEN Ramp_Decel_Rate       := 1.0;   END_IF; (* Gia tốc giảm tốc (D608) *)
IF Decel_Distance_Meters <= 0.0 THEN Decel_Distance_Meters := 50.0;  END_IF; (* Khoảng cách hãm dừng (m) *)

(* ---------------------------------------------------------------------------- *)
(* 8. KHỞI TẠO CÀI ĐẶT LỰC CĂNG (TENSION SP - kg/N - REAL) & HỆ SỐ PID         *)
(* ---------------------------------------------------------------------------- *)
IF SP_Tension_T  <= 0.0 THEN SP_Tension_T  := 15.0; END_IF; (* SP Lực căng Thu T: 15.0 kg (D660) *)
IF SP_Tension_X1 <= 0.0 THEN SP_Tension_X1 := 12.0; END_IF; (* SP Lực căng Xả X1: 12.0 kg (D662) *)
IF SP_Tension_M  <= 0.0 THEN SP_Tension_M  := 10.0; END_IF; (* SP Lực căng Xả M:  10.0 kg (D664) *)
IF SP_Tension_U  <= 0.0 THEN SP_Tension_U  := 10.0; END_IF; (* SP Lực căng Xả U:  10.0 kg (D668) *)

(* Hệ số PID cuộn Thu T *)
IF Kp_T <= 0.0 THEN Kp_T := 1.5; END_IF;
IF Ki_T <= 0.0 THEN Ki_T := 0.2; END_IF;
IF Kd_T <= 0.0 THEN Kd_T := 0.1; END_IF;

(* Hệ số PID cuộn Xả X1 *)
IF Kp_X1 <= 0.0 THEN Kp_X1 := 1.2; END_IF;
IF Ki_X1 <= 0.0 THEN Ki_X1 := 0.15; END_IF;
IF Kd_X1 <= 0.0 THEN Kd_X1 := 0.08; END_IF;

(* Hệ số PID cuộn Xả M *)
IF Kp_M <= 0.0 THEN Kp_M := 1.0; END_IF;
IF Ki_M <= 0.0 THEN Ki_M := 0.1; END_IF;
IF Kd_M <= 0.0 THEN Kd_M := 0.05; END_IF;

(* Hệ số PID cuộn Xả U *)
IF Kp_U <= 0.0 THEN Kp_U := 1.0; END_IF;
IF Ki_U <= 0.0 THEN Ki_U := 0.1; END_IF;
IF Kd_U <= 0.0 THEN Kd_U := 0.05; END_IF;

(* ---------------------------------------------------------------------------- *)
(* 9. KHỞI TẠO TORQUE HÃM MIN / MAX VÀ GIỮ DỪNG MÁY (% - REAL)                 *)
(* ---------------------------------------------------------------------------- *)
IF Min_Torque_M          <= 0.0 THEN Min_Torque_M          := 4.0;  END_IF; (* 4.0 % *)
IF Max_Torque_M          <= 0.0 THEN Max_Torque_M          := 20.0; END_IF; (* 20.0 % *)
IF Init_Holding_Torque_M <= 0.0 THEN Init_Holding_Torque_M := 8.0;  END_IF; (* 8.0 % *)

IF Min_Torque_U          <= 0.0 THEN Min_Torque_U          := 5.0;  END_IF; (* 5.0 % *)
IF Max_Torque_U          <= 0.0 THEN Max_Torque_U          := 25.0; END_IF; (* 25.0 % *)
IF Init_Holding_Torque_U <= 0.0 THEN Init_Holding_Torque_U := 10.0; END_IF; (* 10.0 % *)

(* ---------------------------------------------------------------------------- *)
(* 10. KHỞI TẠO HỆ SỐ GAIN CALIB LOADCELL (REAL)                                *)
(* ---------------------------------------------------------------------------- *)
IF Calib_Gain_T  <= 0.0 THEN Calib_Gain_T  := 1.0; END_IF;
IF Calib_Gain_X1 <= 0.0 THEN Calib_Gain_X1 := 1.0; END_IF;
IF Calib_Gain_M  <= 0.0 THEN Calib_Gain_M  := 1.0; END_IF;
IF Calib_Gain_U  <= 0.0 THEN Calib_Gain_U  := 1.0; END_IF;

(* ---------------------------------------------------------------------------- *)
(* 11. CẤU HÌNH LẤY TRUNG BÌNH NỘI TẠI MODULE CC-LINK 68ADV (AJ65VBT-68ADV - TRẠM 1 & 2) *)
(* ---------------------------------------------------------------------------- *)
(* [GIẢI THÍCH CHẾ ĐỘ LẤY TRUNG BÌNH NỘI TẠI TRONG BUFFER MEMORY CỦA MODULE]:   *)
(*                                                                              *)
(* 1. BFM #0 & BFM #1 - CHỌN CHẾ ĐỘ CHO 8 KÊNH ADC:                             *)
(*    - BFM #0: CH1..CH4 (Mỗi kênh 1 Nibble Hex H[CH4][CH3][CH2][CH1])          *)
(*    - BFM #1: CH5..CH8 (Mỗi kênh 1 Nibble Hex H[CH8][CH7][CH6][CH5])          *)
(*    - 16#0 (0): Lấy mẫu tức thời (Sampling Processing - Mặc định)             *)
(*    - 16#1 (1): Trung bình theo Thời Gian (Time Average - Đơn vị: ms)         *)
(*    - 16#2 (2): Trung bình theo Số Lần   (Count Average - Đơn vị: Lần/Mẫu)    *)
(*    - 16#3 (3): Trung bình Trượt (Moving Average - Khuyên dùng cho Loadcell)  *)
(*                                                                              *)
(*    * VÍ DỤ CÀI ĐẶT BFM #0 & #1:                                              *)
(*      + 16#3333 -> Chạy Trung Bình Trượt (Moving Average) cho 4 kênh          *)
(*                                                                              *)
(* 2. BFM #2..#9 - GIÁ TRỊ CÀI ĐẶT CHO TỪNG KÊNH CH1..CH8:                      *)
(*    - Time Average   (Kiểu 1): 20 ~ 5000 (ms)                                 *)
(*    - Count Average  (Kiểu 2): 4 ~ 500 (lần)                                  *)
(*    - Moving Average (Kiểu 3): 4 ~ 60 (mẫu trượt liên tục - Khuyên đặt: 16)   *)
(* ---------------------------------------------------------------------------- *)

(* A. Gán hằng số chế độ lấy trung bình (16#3333 = Moving Average 8 kênh) *)
CCLink_AD_Avg_Mode := 16#3333; (* D860: Hằng số kiểu lấy trung bình trượt CH1..CH4 *)

(* B. Gán hằng số số mẫu trung bình cho từng kênh CH1..CH8 (16 mẫu trượt) *)
CCLink_AD_Avg_CH1 := 16; (* D861: CH1 (Loadcell Thu T - D500)   - 16 mẫu *)
CCLink_AD_Avg_CH2 := 16; (* D862: CH2 (Loadcell Kéo X1 - D501)  - 16 mẫu *)
CCLink_AD_Avg_CH3 := 16; (* D863: CH3 (Loadcell Thắng M - D502) - 16 mẫu *)
CCLink_AD_Avg_CH4 := 16; (* D864: CH4 (Loadcell Xả U - D503)    - 16 mẫu *)

(* C. Gán hằng số cho phép chuyển đổi A/D cả 8 kênh *)
CCLink_AD_Conv_En := 0;  (* D865: Cho phép chuyển đổi toàn bộ kênh *)
END_PROGRAM

// device comments not shown above
M1104  ; Remote Input X0 (St4)
M1105  ; Remote Input X1 (St4)
M1106  ; Remote Input X2 (St4)
M1107  ; Remote Input X3 (St4)
M1108  ; Remote Input X4 (St4)
M1109  ; Remote Input X5 (St4)
M1110  ; Remote Input X6 (St4)
M1111  ; Remote Input X7 (St4)
M1304  ; Servo ON Truc Thu T (Y8)
M1305  ; Servo ON Truc Xa X1 (Y9)
M1306  ; Servo ON Truc Master X2 (YA)
M1307  ; Servo ON Truc Ghep Ms (YB)
M1308  ; Servo ON Truc Trang Dau S (YC)
M1309  ; Solenoid Valve Pen 1 (YD)
M1310  ; Solenoid Valve Pen 2 (YE)
D524  ; DAC CH1: Speed Thu T
D525  ; DAC CH2: Torque Thu T
D526  ; DAC CH3: Speed Xa X1
D527  ; DAC CH4: Speed Master X2
D528  ; DAC CH5: Speed Ghep Ms
X50  ; "X","50","Sensor tiem can dem vo
X51  ; "X","51","Sensor tiem can dem vo
X52  ; "X","52","Nut nhan START vat ly
X53  ; "X","53","Nut nhan STOP vat ly (
X54  ; "X","54","Nut nhan INC Tang toc
X55  ; "X","55","Nut nhan DEC Giam toc
X56  ; "X","56","Nut Toggle Pen 1 vat l
X57  ; "X","57","Nut Toggle Pen 2 vat l
X58  ; "X","58","Cong tac Giu Torque M
X59  ; "X","59","Cong tac Giu Torque U
X5A  ; "X","5A","Cong tac Rua may bo ch
X5B  ; "X","5B","Cong tac Rua may bo ch
X5C  ; "X","5C","Nut nhan co BO CHAM NO
M1208  ; Cho phép chuyển đổi A/D Trạm 1 (
M1240  ; Cho phép chuyển đổi D/A Trạm 2 (
M1311  ; Du phong / Bao loi (YF)
D529  ; DAC CH6: Torque Ghep Ms
D530  ; DAC CH7: Speed Trang Dau S
D531  ; DAC CH8: Speed Xa U
